130:(* Wait for Finishing movement *)
		IF 	(MoveWorkStored AND WorkPosition) OR
			(MoveInitStored AND InitPosition)	THEN
			WorkingStep:=140;
		END_IF
140:(* Reset Coils if necessary *)
		IF  sInit.KindOfValve='B' AND
			(	( NoOfWorkSensors>0 AND MoveWorkStored) OR
				( NoOfInitSensors>0 AND MoveInitStored) ) THEN
			CoilA:=FALSE;
			CoilB:=FALSE;
			WorkingStep:=1000;
		ELSE
			WorkingStep:=1000;
		END_IF
999: (* State Error *)
		State:=STATE_ERROR;
1000: (* State OK *)
		State:=STATE_OK;
		TimerTimeOut.Start:=FALSE;
		IF 	NOT MoveWork AND	NOT MoveInit OR
			MoveInit AND MoveWorkStored OR
			MoveWork AND MoveInitStored THEN
			WorkingStep:=0;
		END_IF
	END_CASE
	(*--------------------------------------------------------------------
		Handle Timeout
  --------------------------------------------------------------------*)
	IF TimerTimeOut.Timeout THEN
		State:=STATE_TIMEOUT;
		FB_ReadXmlLineMsg.ID:='timeout';
		Error.No:=1;
		Error.Text:=sInit.InstName;
		Error.Text:=CONCAT(Error.Text,': ');
		Error.Text:=CONCAT(Error.Text,sInit.Description);
		Error.Text:=CONCAT(Error.Text,' - ');
		Error.Text:=CONCAT(Error.Text,FB_ReadXmlLineMsg.Text);

		(* Set Flags to Raise Error in ValveSensor Object *)
		IF 	NoOfInitSensors>0 THEN
			FOR IdxInit:=1 TO NoOfInitSensors DO
				ValveInitOut[IdxInit].SignalHiExpected:=MoveInitStored;
				ValveInitOut[IdxInit].SignalLoExpected:=MoveWorkStored;
			END_FOR
		END_IF
		IF 	NoOfWorkSensors>0 THEN
			FOR IdxWork:=1 TO NoOfWorkSensors DO
				ValveWorkOut[IdxWork].SignalHiExpected:=MoveWorkStored;
				ValveWorkOut[IdxWork].SignalLoExpected:=MoveInitStored;
			END_FOR
		END_IF
	ELSE
		(* Reseet Flags to Raise Error in ValveSensor Object *)
		IF 	NoOfInitSensors>0 THEN
			FOR IdxInit:=1 TO NoOfInitSensors DO
				ValveInitOut[IdxInit].SignalHiExpected:=FALSE;
				ValveInitOut[IdxInit].SignalLoExpected:=FALSE;
			END_FOR
		END_IF
		IF 	NoOfWorkSensors>0 THEN
			FOR IdxWork:=1 TO NoOfWorkSensors DO
				ValveWorkOut[IdxWork].SignalHiExpected:=FALSE;
				ValveWorkOut[IdxWork].SignalLoExpected:=FALSE;
			END_FOR
		END_IF
	END_IF
	(*--------------------------------------------------------------------
		Handle unallowed Signalchange without Movecommand
  --------------------------------------------------------------------*)
	IF 	State=State_Wait AND
		NOT sInit.DisableSignalMonitoring THEN
		(* Set Flags to Raise Error in ValveSensor Object *)
		IF  	(MoveInitStored AND NOT InitPosition) OR
			(MoveWorkStored AND NOT WorkPosition)	THEN
			State:=STATE_ERROR;
			FB_ReadXmlLineMsg.ID:='SensorFault';
			Error.No:=1;
			Error.Text:=sInit.InstName;
			Error.Text:=CONCAT(Error.Text,': ');
			Error.Text:=CONCAT(Error.Text,sInit.Description);
			Error.Text:=CONCAT(Error.Text,' - ');
			Error.Text:=CONCAT(Error.Text, FB_ReadXmlLineMsg.Text);

			IF 	NoOfInitSensors>0 THEN
				FOR IdxInit:=1 TO NoOfInitSensors DO
					ValveInitOut[IdxInit].SignalHiExpected:=MoveInitStored;
					ValveInitOut[IdxInit].SignalLoExpected:=MoveWorkStored;
				END_FOR
			END_IF
			IF 	NoOfWorkSensors>0 THEN
				FOR IdxWork:=1 TO NoOfWorkSensors DO
					ValveWorkOut[IdxWork].SignalHiExpected:=MoveWorkStored;
					ValveWorkOut[IdxWork].SignalLoExpected:=MoveInitStored;
				END_FOR
			END_IF
		END_IF

	END_IF
	(*--------------------------------------------------------------------
		Call Timers
  --------------------------------------------------------------------*)
	TimerTimeOut(MTime:=sInit.MaxTime);
	DampBothTimer(PT:=DINT_TO_TIME(sInit.DampBothTime));
	(*--------------------------------------------------------------------
		Updating processtime (if State_RUN, STATE_TIMEOUT, STATE_RESETS, or STATE_STOPPED)
  --------------------------------------------------------------------*)
	IF	(State=State_RUN OR
		State=STATE_TIMEOUT OR
		State=STATE_RESETS OR
		State=STATE_STOPPED) AND
		sInit.MaxTime<>0 AND
		 ( NoOfInitSensors<>0 OR NoOfWorkSensors<>0)	THEN
		ProcessTime:=TimerTimeOut.PTime;
	END_IF
(*--------------------------------------------------------------------
	HomePosition
  --------------------------------------------------------------------*)

IF	sVisu.Description <> '' THEN
	CASE	sInit.HomePosDefine OF

	HOME_INIT:
		HomePosition:=InitPosition AND NOT WorkPosition AND (sInit.KindOfValve<>'2G' OR CoilBState);
	HOME_WORK:
		HomePosition:=WorkPosition AND NOT InitPosition AND (sInit.KindOfValve<>'2G' OR CoilAState);
	HOME_BOTH:
		HomePosition:=WorkPosition OR InitPosition;
	HOME_ALWAYS:
		HomePosition:=TRUE;
	ELSE
		HomePosition:=FALSE;
	END_CASE


(* Generating home position*)
	IF 	NOT HomePosition THEN
		ListHomeNOK(InstName:=sInit.InstName,Description:=FB_ReadXmlLineConf.Text);
	END_IF

	(* Object-homeposition concat with mainhomeposition *)
	gHomeOk:=gHomeOk AND HomePosition;
END_IF
(*------------------------------------------------------------------
	Update Visu
  ------------------------------------------------------------------*)
	sVisu.InstName:=sInit.InstName;

	sVisu.ProcessTime:=ProcessTime;
	sVisu.HomePosition:=HomePosition;
	sVisu.CoilA:=CoilA;
	sVisu.CoilB:=CoilB;
	sVisu.NoOfInitSensors:=NoOfInitSensors;
	sVisu.NoOfWorkSensors:=NoOfWorkSensors;
	sVisu.NoOfValveCoils:=NoOfValveCoils;

	sVisu.SAInitPosName:=SensorInitIn[1].SensorName;
	sVisu.SBInitPosName:=SensorInitIn[2].SensorName;
	sVisu.SCInitPosName:=SensorInitIn[3].SensorName;
	sVisu.SDInitPosName:=SensorInitIn[4].SensorName;
	sVisu.SEInitPosName:=SensorInitIn[5].SensorName;
	sVisu.SAWorkPosName:=SensorWorkIn[1].SensorName;
	sVisu.SBWorkPosName:=SensorWorkIn[2].SensorName;
	sVisu.SCWorkPosName:=SensorWorkIn[3].SensorName;
	sVisu.SDWorkPosName:=SensorWorkIn[4].SensorName;
	sVisu.SEWorkPosName:=SensorWorkIn[5].SensorName;

	sVisu.AInitPosition:=SensorInitIn[1].SensorSignal;
	sVisu.BInitPosition:=SensorInitIn[2].SensorSignal;
	sVisu.CInitPosition:=SensorInitIn[3].SensorSignal;
	sVisu.DInitPosition:=SensorInitIn[4].SensorSignal;
	sVisu.EInitPosition:=SensorInitIn[5].SensorSignal;
	sVisu.AWorkPosition:=SensorWorkIn[1].SensorSignal;
	sVisu.BWorkPosition:=SensorWorkIn[2].SensorSignal;
	sVisu.CWorkPosition:=SensorWorkIn[3].SensorSignal;
	sVisu.DWorkPosition:=SensorWorkIn[4].SensorSignal;
	sVisu.EWorkPosition:=SensorWorkIn[5].SensorSignal;

(*------------------------------------------------------------------
	Reset-Handling
  ------------------------------------------------------------------*)
IF 	Reset THEN
	State:=STATE_RESETS;
	WorkingStep:=0;
	ProcessTime:=0;
	TimerTimeOut.Start:=FALSE;
	DampBothTimer.IN:=FALSE;
	CoilA:=FALSE;
	CoilB:=FALSE;
	MoveWorkStored:=FALSE;
	MoveInitStored:=FALSE;
END_IF

(*------------------------------------------------------------------
	Error-Handling
  ------------------------------------------------------------------*)
ErrorElapsed(CLK:= Error.Text<>'');
IF ErrorElapsed.Q THEN
	Error.DateTime:=gVarDTSystemtime;
END_IF

IF Error.Text<>''	AND ST_Lng.b_EndChangeLng THEN
	Error.Typ:=0;
	(*Error.DateTime:=;*)
	ErrorHandler.AddError(
			ErrorToAdd:=Error,
			sVisu:=Visu.ErrorHandler);
END_IF

IF 	NOT Enable AND ModeSelect.Mode=MODE_MANUAL AND
	Error.Text='' AND strAnlayse<>''THEN

	strAnlayse:=CONCAT(' +++ gesperrt durch : ',strAnlayse);

	LaufschriftAnalyse(
	N:= 40,
	StepWidth:=1,
	PT:= t#100ms ,
	Text:= strAnlayse,
	Display=>sVisu.ErrorString );

	strAnlayse:='';
ELSE
	IF Error.Text<>'' THEN
		TempString:=CONCAT(' --- ',Error.Text);
		LaufschriftObj(
		N:= 40,
		StepWidth:=1,
		PT:= t#100ms ,
		Text:= TempString,
		Display=>sVisu.ErrorString );
	ELSE
		sVisu.ErrorString:='';
	END_IF
END_IF

(*------------------------------------------------------------------
	Reset Inputs
  ------------------------------------------------------------------*)
MoveWork		:=FALSE; 				(* Move to Workposition *)
MoveInit		:=FALSE;				(* Move to Initposition *)
Enable			:=FALSE; 				(* Enables the operations on the valve *)
Reset			:=FALSE; 				(* switch for resetting the object *)

sVisu.InstName:=sInit.InstName;
sVisu.BitName:=sInit.BitName;
sVisu.BtnMoveWork.Text:=sInit.WorkDescription;
sVisu.BtnMoveInit.Text:=sInit.InitDescription;
sVisu.ErrorPresent:=Error.Text<>'';

FB_ReadXmlLineConf(
	Prefix:= 'CONFIG',
	ID:= sInit.InstName,
	File:= 'CONFIG.xml',
	Text=> sVisu.Description );

FB_ReadXmlLineMsg(
	Prefix:= 'MSG',
	ID:= ,
	File:= 'MSG.xml',
	Text=>);


IF 	State = STATE_ERROR THEN
	Error.Text:=sInit.InstName;
	Error.Text:=CONCAT(Error.Text,': ');
	Error.Text:=CONCAT(Error.Text,sInit.Description);
	Error.Text:=CONCAT(Error.Text,' - ');
	Error.Text:=CONCAT(Error.Text,FB_ReadXmlLineMsg.Text);
END_IF
END_FUNCTION_BLOCK
ACTION AddInitSensor:
NoOfInitSensors:=NoOfInitSensors+1;
END_ACTION
ACTION AddWorkSensor:
NoOfWorkSensors:=NoOfWorkSensors+1;
END_ACTION

(* POU System/HelpFunctions/CheckProcTime, ST *)
FUNCTION_BLOCK CheckProcTime
VAR_OUTPUT
	PTime		: DINT;	(* Time since start of the timer *)
	Timeout		: BOOL; (* Flag if Timeout occured *)
END_VAR
VAR_INPUT
	MTime		: DINT;	(* Time to timeout *)
	Start		: BOOL;	(* True starts the Timer, False resets *)
END_VAR
VAR
	TONT		: TON;	(* Timer counting Timer *)
END_VAR
(* Start Timer if Start is True.
Stop Timer ,if Start is false.
Timer maximal counting to two hours. *)
TONT(IN:=Start,PT:=T#2h);

(* Updating the Processtime PTime. You get it if you change the output ET of TONT to DWORD.. *)
PTime:=TIME_TO_DWORD(TONT.ET);

(* Setting output Timeout
No Timeout IF Timer stopped OR mtime > ptime*)
IF 	MTime > PTime OR NOT Start THEN
	Timeout:=FALSE;
ELSE
	Timeout:=TRUE;
END_IF
END_FUNCTION_BLOCK

(* POU zLibrary/_HelpFunctions/FB_Laufschrift, ST *)
FUNCTION_BLOCK FB_Laufschrift
VAR_INPUT
	N 						:INT; (* Max output Stringlength *)
	StepWidth				:INT:=1;
	PT 						:TIME;
	Text 					:STRING; (* Original String *)
END_VAR
VAR_OUTPUT
	Display 					:STRING(255); (* Output String *)
END_VAR
VAR
	delay 					:TP;
	TempOutputString		:STRING(255);
	TempInputText			:STRING(255);
	step 					:INT;
END_VAR
(* generate next ticker when delay is low *)
IF 	N < LEN(text) THEN
	IF 	NOT delay.Q THEN
		(* increase step for next tick *)
		TempInputText:=text;
		step := step + StepWidth;

		IF step > LEN(TempInputText) THEN
			step := 1;
		END_IF

		(* extract dispay from text *)
		TempOutputString := MID(TempInputText, N, step);

		IF 	LEN(TempOutputString)<N THEN
			TempOutputString:=CONCAT(TempOutputString,TempInputText);
			TempOutputString:=LEFT(TempOutputString,N);
			Display:=TempOutputString;
		ELSE
			Display:=TempOutputString;
		END_IF
		(* set delay timer for next tick *)
		delay(IN := TRUE, PT := PT);
	ELSE
		(* execute delay timer *)
		delay(in := FALSE);
	END_IF
ELSE
	display := text;
END_IF
END_FUNCTION_BLOCK

(* POU zLibrary/Valve/FB_ValveSensor, ST *)
FUNCTION_BLOCK FB_ValveSensor
VAR_INPUT
	ValveObject					: POINTER TO FB_Valve;		(* Pointer to declared Valve Instance *)
	sInit							: sValveSensorInit; 				(* Intialisation Informations e.g. Object Name *)
END_VAR
VAR_IN_OUT

END_VAR
VAR_OUTPUT
END_VAR
VAR
	ValveSensor	 			AT %I* :	BOOL; 					(* Sensor A InitPosition *)

	(* Sensor Handling *)
	ValveOut					: sValveSensor_ValveOut; 		(* Signals from Valve Object *)
	SensorOut					: sValveSensor_SensorOut;		(* Signals to Valve Object *)

	ValveSensorNo				: DINT; 							(* Number of Sensor given from ValveObject *)

	sVisuValveDummy			: sValveVisu; 					(* Dummy struct for Calling Action from Valve Object  *)

(* Init Handling *)
	InitState						: BOOL :=	FALSE;				(* Internal State for initialising *)
	InitStep						: INT;							(* Init Step StateMachine *)

(*  Error Handling *)
	Error						: ErrorStruct;						(* Local Error Struct *)
	ErrorElapsed				: R_TRIG;						(* Flag to Store Systemtime in Errorstruct when the error raising *)

	FB_ReadXmlLineConf		: FB_ReadXmlLine;
	FB_ReadXmlLineMsg		: FB_ReadXmlLine;
END_VAR
IF 	NOT InitState THEN
	CASE InitStep OF
	0: (* Init Instance *)
			InitStep:=100;

	100: (* Init Done *)

		IF	ValveSensorNo=0 THEN
			IF sInit.SensorType=sValveSensorType_INIT	THEN
		   		ValveObject^.AddInitSensor(sVisu:=sVisuValveDummy);
				ValveSensorNo:=ValveObject^.NoOfInitSensors;
			ELSE
		   		ValveObject^.AddWorkSensor(sVisu:=sVisuValveDummy);
				ValveSensorNo:=ValveObject^.NoOfWorkSensors;
			END_IF

			SensorOut.SensorName:=sInit.BitName;
			SensorOut.SensorType:=sInit.SensorType;

		END_IF

		InitState:=TRUE;
	END_CASE


ELSE
	(* Init State OK *)
	Error.No:=0;
	Error.Text:='';

	IF 	sInit.SensorType=sValveSensorType_INIT	THEN
		ValveOut:=ValveObject^.ValveInitOut[ValveSensorNo];
	ELSE
		ValveOut:=ValveObject^.ValveWorkOut[ValveSensorNo];
	END_IF

	(* Generate Errors  *)

	(* Check Signal Hi *)
	IF 	ValveOut.SignalHiExpected AND
		NOT ValveSensor	THEN
	  	Error.No:=1;
(*		Error.Text:=CONCAT(ValveObject^.sInit.InstName,' - ');*)
		FB_ReadXmlLineMsg.ID:='SensorFaultNotHigh';
		Error.Text:=CONCAT(Error.Text,sInit.InstName);
		Error.Text:=CONCAT(Error.Text,' :');
		Error.Text:=CONCAT(Error.Text,FB_ReadXmlLineConf.Text);
		Error.Text:=CONCAT(Error.Text,' - ');
		Error.Text:=CONCAT(Error.Text,FB_ReadXmlLineMsg.Text);

	END_IF


	(* Check Signal Low *)
	IF 	ValveOut.SignalLoExpected AND
		ValveSensor THEN
	  	Error.No:=1;
(*		Error.Text:=CONCAT(ValveObject^.sInit.InstName,' - ');*)
		FB_ReadXmlLineMsg.ID:='SensorFaultNotLow';
		Error.Text:=CONCAT(Error.Text,sInit.InstName);
		Error.Text:=CONCAT(Error.Text,' :');
		Error.Text:=CONCAT(Error.Text,FB_ReadXmlLineConf.Text);
		Error.Text:=CONCAT(Error.Text,' - ');
		Error.Text:=CONCAT(Error.Text,FB_ReadXmlLineMsg.Text);
	END_IF

	(* Write Sensor stete in local out Structure *)
	SensorOut.SensorSignal:=ValveSensor;

	(* Give local "out structure" to Valve object *)
	IF 	sInit.SensorType=sValveSensorType_INIT THEN
		ValveObject^.SensorInitIn[ValveSensorNo]:=SensorOut;
	ELSE
		ValveObject^.SensorWorkIn[ValveSensorNo]:=SensorOut;
	END_IF

END_IF

(*------------------------------------------------------------------
	Error-Handling
  ------------------------------------------------------------------*)

ErrorElapsed(CLK:= Error.Text<>'');
IF 	ErrorElapsed.Q THEN
	Error.DateTime:=gVarDTSystemtime;
END_IF

IF Error.Text<>''	AND ST_Lng.b_EndChangeLng THEN
	Error.Typ:=0;
	ErrorHandler.AddError(
				ErrorToAdd:=Error,
				sVisu:=Visu.ErrorHandler);
END_IF

(*------------------------------------------------------------------
	Language-Handling
  ------------------------------------------------------------------*)

FB_ReadXmlLineConf(
	Prefix:= 'CONFIG',
	ID:= sInit.InstName,
	File:= 'CONFIG.xml',
	Text=> );


FB_ReadXmlLineMsg(
	Prefix:= 'MSG',
	ID:= ,
	File:= 'MSG.xml',
	Text=>);

IF 	Error.Text<>'' THEN
	Error.Text:=CONCAT(Error.Text,sInit.InstName);
	Error.Text:=CONCAT(Error.Text,' :');
	Error.Text:=CONCAT(Error.Text,FB_ReadXmlLineConf.Text);
	Error.Text:=CONCAT(Error.Text,' - ');
	Error.Text:=CONCAT(Error.Text,FB_ReadXmlLineMsg.Text);
END_IF
END_FUNCTION_BLOCK

(* POU zLibrary/AnaIn/FB_AnaInDint, ST *)
FUNCTION_BLOCK FB_AnaInDint
VAR_INPUT
	sInit					:sAnaInInit;	(* Initializingvalues to the Instance *)
END_VAR
VAR_OUTPUT
	State					:StateObject;	(* State of the object *)
	HomePosition			:BOOL;			(* object in home-position*)
	Value					:REAL;
END_VAR
VAR_IN_OUT
	sVisu					:sAnaInVisu;
END_VAR
VAR
	AnaInValue		AT %I* 	:DINT;			(* Ana in value *)

	Error					:ErrorStruct;
	TempErrorText			:STRING(255);
	InitState				:BOOL:=FALSE;	(* Internal State for initialising *)

	diffSource				:REAL;
	diffTarget				:REAL;

	FB_ReadXmlLineConf		:FB_ReadXmlLine;
	FB_ReadXmlLineMsg		:FB_ReadXmlLine;
END_VAR
Error.No:=0;
Error.Text:='';

(*------------------------------------------------------------------
	Initialization
  ------------------------------------------------------------------*)
IF  NOT InitState THEN
	InitState:=TRUE;

	(* Check instance name *)
	IF sInit.InstName=''THEN
		InitState:=FALSE;
		State:=STATE_ERROR;
		FB_ReadXmlLineMsg.ID:='InstNameNotDefined';

		TempErrorText:=sInit.BitInName;
		TempErrorText:=CONCAT(TempErrorText,' :');
		TempErrorText:=CONCAT(TempErrorText,sVisu.Description);
  		TempErrorText:=CONCAT(TempErrorText,' -> ');
		TempErrorText:=CONCAT(TempErrorText,FB_ReadXmlLineMsg.Text);
		Error.No:=4;
		(*Error.Text:='InstName not defined';*)
	(*CheckDescription*)
	ELSIF
		sInit.Description=''THEN
		InitState:=FALSE;
		State:=STATE_ERROR;
		FB_ReadXmlLineMsg.ID:='DescriptionNotDefined';

		TempErrorText:=sInit.BitInName;
		TempErrorText:=CONCAT(TempErrorText,' :');
		TempErrorText:=CONCAT(TempErrorText,sVisu.Description);
  		TempErrorText:=CONCAT(TempErrorText,' -> ');
		TempErrorText:=CONCAT(TempErrorText,FB_ReadXmlLineMsg.Text);
		Error.No:=4;
		(*Error.Text:='Description not defined';*)
	END_IF

	sVisu.InstName		:= sInit.InstName;
	sVisu.Description	:= sInit.Description;
	sVisu.ErrorString	:= Error.Text;
END_IF

(* Add InitState to Global-Init-State to collect all Objects *)
gInitCollect:=gInitCollect AND InitState;

IF 	InitState THEN
	diffSource := sinit.ScalingSensorValueMax - sinit.ScalingSensorValueMin;
  	diffTarget := sinit.ScalingOutputValueMax - sinit.ScalingOutputValueMin;
 	(*Value := (((AnaInValue-sinit.ScalingOutputValueMin)/diffSource)*diffTarget)+sinit.ScalingOutputValueMin;*)
 	Value :=  (AnaInValue- sinit.ScalingSensorValueMin) / (diffSource  / diffTarget) ;

	sVisu.AnaInValue:=Value;

END_IF
(* ------------------------------------------------------------------------------------------ *)
(* ---------------- LANGUAGE auslesen aus der XML Datei-------- *)
(* ------------------------------------------------------------------------------------------ *)
sVisu.BitInName:=sInit.BitInName;
sVisu.InstName:=sInit.InstName;
sVisu.ErrorPresent:=Error.Text<>'';

FB_ReadXmlLineConf(
	Prefix:= 'CONFIG',
	ID:= sInit.InstName,
	File:= 'CONFIG.xml',
	Text=> sVisu.Description  );


FB_ReadXmlLineMsg(
	Prefix:= 'MSG',
	ID:= ,
	File:= 'MSG.xml',
	Text=>);

IF 	State = STATE_ERROR THEN
	TempErrorText:=sInit.BitInName;
	TempErrorText:=CONCAT(TempErrorText,' :');
	TempErrorText:=CONCAT(TempErrorText,sVisu.Description);
	TempErrorText:=CONCAT(TempErrorText,' -> ');
	TempErrorText:=CONCAT(TempErrorText,FB_ReadXmlLineMsg.Text);
END_IF
END_FUNCTION_BLOCK

(* POU zLibrary/AnaIn/FB_Encoder, ST *)
FUNCTION_BLOCK FB_Encoder
VAR_INPUT
	sInit					:sEncoderInit;	(* Initializingvalues to the Instance *)
	Reset					:BOOL;
END_VAR
VAR_OUTPUT
	State					:StateObject;	(* State of the object *)
	rpmValue			: LREAL;		(* rpm *)
	posValue			: LREAL;		(* mm *)
	Drehrichtung		: enum_Drehrichtung;
END_VAR
VAR_IN_OUT
	sVisu				:sEncoderVisu;
END_VAR
VAR

	Error					:ErrorStruct;
	TempErrorText			:STRING(255);
	ErrorElapsed			:BOOL;
	LaufschriftErrh			:FB_Laufschrift;
	LaufschriftObj			:FB_Laufschrift_STR255;
	InitState				:BOOL:=FALSE;	(* Internal State for initialising *)



	FB_ReadXmlLineConf		:FB_ReadXmlLine;
	FB_ReadXmlLineMsg		:FB_ReadXmlLine;
END_VAR


(*==================================================================*)
VAR_OUTPUT

END_VAR

VAR
	fb_ton_Reset		: TON;
	fb_ton_steht		: TON;
	fb_ton_dreht		: TON;

	fb_rTrigReset		: R_TRIG;
	fb_rTrigUnderflow		: R_TRIG;
	fb_rTrigOverflow		: R_TRIG;

	i_count_ueberlauf		: DINT;		(* +- 64bit *)
	lr_xBit		: LREAL;
	lr_rpmHelp	: LREAL;	(*°*)

	
	e_Value					AT %I* : UINT;		(* 65535 *)
	e_CountUnderflow		AT %I* : BOOL;
	e_CountOverflow			AT %I* : BOOL;
	a_CountReset			AT %Q* : BOOL;

END_VAR
VAR CONSTANT



END_VAR
Error.No:=0;
Error.Text:='';

(*------------------------------------------------------------------
	Initialization
  ------------------------------------------------------------------*)
IF  NOT InitState THEN
	InitState:=TRUE;
	State:=STATE_OK;
	(* Check instance name *)
	IF 	sInit.InstName=''THEN
		InitState:=FALSE;
		State:=STATE_ERROR;
		FB_ReadXmlLineMsg.ID:='InstNameNotDefined';

		TempErrorText:=sInit.BitInName;
		TempErrorText:=CONCAT(TempErrorText,' :');
		TempErrorText:=CONCAT(TempErrorText,sVisu.Description);
  		TempErrorText:=CONCAT(TempErrorText,' -> ');
		TempErrorText:=CONCAT(TempErrorText,FB_ReadXmlLineMsg.Text);
		Error.No:=4;
	(*CheckDescription*)
	ELSIF
		sInit.Description=''THEN
		InitState:=FALSE;
		State:=STATE_ERROR;
		FB_ReadXmlLineMsg.ID:='DescriptionNotDefined';

		TempErrorText:=sInit.BitInName;
		TempErrorText:=CONCAT(TempErrorText,' :');
		TempErrorText:=CONCAT(TempErrorText,sVisu.Description);
  		TempErrorText:=CONCAT(TempErrorText,' -> ');
		TempErrorText:=CONCAT(TempErrorText,FB_ReadXmlLineMsg.Text);
		Error.No:=4;
	ELSIF
		sInit.i_InkProRpm=0THEN
		InitState:=FALSE;
		State:=STATE_ERROR;
		FB_ReadXmlLineMsg.ID:='InkProRpmNotDefined';

		TempErrorText:=sInit.BitInName;
		TempErrorText:=CONCAT(TempErrorText,' :');
		TempErrorText:=CONCAT(TempErrorText,sVisu.Description);
  		TempErrorText:=CONCAT(TempErrorText,' -> ');
		TempErrorText:=CONCAT(TempErrorText,FB_ReadXmlLineMsg.Text);
		Error.No:=4;
	END_IF

END_IF

(* Add InitState to Global-Init-State to collect all Objects *)
gInitCollect:=gInitCollect AND InitState;

(*==================================================================*)
IF  InitState THEN
	(* Drehrichtung ermitteln *)
	fb_ton_steht(PT:=T#50MS);
	IF	lr_rpmHelp > rpmValue - 0.0001 AND
		lr_rpmHelp < rpmValue + 0.0001 THEN
		fb_ton_steht.IN:=TRUE;
		IF	fb_ton_steht.Q THEN
			Drehrichtung:= STEHT;
		END_IF
	ELSIF
		lr_rpmHelp < rpmValue THEN
		fb_ton_steht.IN:=FALSE;
		Drehrichtung:= VORWAERTS;
	ELSIF
		lr_rpmHelp > rpmValue THEN
		fb_ton_steht.IN:=FALSE;
		Drehrichtung:= RUECKWAERTS;
	END_IF
	lr_rpmHelp:=rpmValue;
	
	(* Encoderüberlauf*)
	fb_rTrigUnderflow(CLK:= e_CountUnderflow);
	fb_rTrigOverflow(CLK:= e_CountOverflow);
	IF 	fb_rTrigUnderflow.Q THEN
		i_count_ueberlauf:=i_count_ueberlauf - 1;
	ELSIF
		fb_rTrigOverflow.Q THEN
		i_count_ueberlauf:=i_count_ueberlauf + 1;
	END_IF

	(* bei Reset Nullen *)
	fb_ton_Reset(IN:=Reset , PT:= T#300MS , Q=> , ET=> );
	a_CountReset:=Reset OR sVisu.Reset;
	fb_rTrigReset(CLK:=fb_ton_Reset.Q, );
	IF	fb_rTrigReset.Q THEN
		Reset:=FALSE;
	END_IF

	(* aktuelle Position *)
	IF	e_Value <> 0 THEN
		lr_xBit:=EXPT(2,16);												(* 16 bit=65535  Inkremente Encoder*)
		rpmValue:= e_Value + (lr_xBit * DINT_TO_LREAL(i_count_ueberlauf));	(* Inkremente*)
		rpmValue:= rpmValue / sInit.i_InkProRpm;							(* Umdrehungen in Grad*)
	ELSE
		rpmValue:= 0;
		i_count_ueberlauf:=0;
	END_IF
	IF	sInit.lr_LaengeProRpm > 0 THEN
		posValue:= rpmValue * sInit.lr_LaengeProRpm;					(* Strecke in mm*)
	ELSE
		posValue:= 0;													(* Strecke in mm*)
	END_IF

	sVisu.posValue:=posValue;
	sVisu.rpmValue:=rpmValue;
	sVisu.Drehrichtung:=Drehrichtung;
END_IF
(* ------------------------------------------------------------------------------------------ *)
(* ---------------- LANGUAGE auslesen aus der XML Datei-------- *)
(* ------------------------------------------------------------------------------------------ *)
sVisu.BitInName:=sInit.BitInName;
sVisu.InstName:=sInit.InstName;
sVisu.ErrorPresent:=Error.Text<>'';

(*  *)
IF 	State=STATE_ERROR AND
	NOT ErrorElapsed THEN
	ErrorElapsed:=TRUE;
	Error.DateTime:=gVarDTSystemtime;
ELSIF
	State<>STATE_ERROR THEN
	ErrorElapsed:=FALSE;
	TempErrorText:='';
END_IF;

IF 	Error.Text<>'' AND
	ST_Lng.b_EndChangeLng THEN
	(*Error.DateTime:=;*)
	Error.Typ:=0;
	ErrorHandler.AddError(ErrorToAdd:=Error,
	sVisu:=Visu.ErrorHandler);
END_IF


FB_ReadXmlLineConf(
	Prefix:= 'CONFIG',
	ID:= sInit.InstName,
	File:= 'CONFIG.xml',
	Text=> sVisu.Description  );

FB_ReadXmlLineMsg(
	Prefix:= 'MSG',
	ID:= ,
	File:= 'MSG.xml',
	Text=>);

IF 	State = STATE_ERROR THEN
	TempErrorText:=sInit.BitInName;
	TempErrorText:=CONCAT(TempErrorText,' :');
	TempErrorText:=CONCAT(TempErrorText,sVisu.Description);
	TempErrorText:=CONCAT(TempErrorText,' -> ');
	TempErrorText:=CONCAT(TempErrorText,FB_ReadXmlLineMsg.Text);
END_IF


LaufschriftErrh(
N:= 160,
StepWidth:=1,
PT:= t#100ms ,
Text:= TempErrorText,
Display=>Error.Text );

LaufschriftObj(
N:= 40,
StepWidth:=1,
PT:= t#100ms ,
Text:= TempErrorText,
Display=>sVisu.ErrorString );
END_FUNCTION_BLOCK

(* POU zLibrary/DigIn/FB_DigIn, ST *)
FUNCTION_BLOCK FB_DigIn

VAR_OUTPUT
	State						: StateObject;	(* State of the object *)
	HomePosition				: BOOL;			(* object in home-position*)
	SignalIn						: BOOL;			(* Static signal of digital input *)
	SignalInDelayed				: BOOL;			(* Static signal of digital input but with on and of delay times *)
END_VAR
VAR_INPUT
	CheckSignalHigh			: BOOL;		 	(* Signal check  HIGH *)
	CheckSignalLow			: BOOL;		 	(* Signal check  LOW  *)

	Reset						: BOOL;			(* switch for resetting the control *)

	SFCCurrentStep				: STRING(40);	(* aktually step in the order of events *)
	SFCCurrentPOU				: STRING(40);	(* Name of the order of events*)

	sInit						: sDigInInit;		(* Initializingvalues to the Instance *)
END_VAR
VAR_IN_OUT
	sVisu						: sDigInVisu;
END_VAR
VAR
	BitInToCheck				AT %I* :BOOL;		(* Bit input signal to check *)

	ProcessTime					: DINT;					(* Counts the time in steps of 100ms since starting operation *)

	TimerTimeOut				: CheckProcTime;		(* Timer generates timeout signal *)
	Error						: ErrorStruct;
	ErrorElapsed				: BOOL;
	TempErrorText				: STRING(255);
	HomePositionInfo			: DINT;							(* missing to home posistion *)
	ResetIntern					: BOOL;							(* Internal reset signal *)


	BtnReset					: VisuButton;			(* Manage button *)

	StateOK_CycleFlag			: BOOL;

	FirstCheckCycle				:  R_TRIG;

	IputOnDelayTime				: TON;
	IputOffDelayTime			: TOF;

	(* --------------------------------------------------------------------------------- *)
	(*         Internal Variables	Visu				                                           *)
	(* --------------------------------------------------------------------------------- *)
	LaufschriftErrh				:FB_Laufschrift;
	LaufschriftObj				:FB_Laufschrift;

	FB_ReadXmlLineConf		:FB_ReadXmlLine;
	FB_ReadXmlLineMsg		:FB_ReadXmlLine;

END_VAR
Error.No:=0;
Error.Text:='';
TempErrorText:='';

(*------------------------------------------------------------------
	Initialization
  ------------------------------------------------------------------*)


(* Add InitState to Global-Init-State to collect all Objects *)
gInitCollect:=gInitCollect ;

IF gInitOk THEN

StateOK_CycleFlag := State=State_ok;


(*------------------------------------------------------------------
	Show and Read Buttons
  ------------------------------------------------------------------*)

BtnReset(	Button:=sVisu.BtnReset,
					Enable:=TRUE ,
					Visible:=ModeSelect.Mode=MODE_MANUAL,
					TextOn:='Reset',
					TextOff:='Reset',
					PressedExt:=FALSE ,
					StateOn:= FALSE ,
					);

	(*------------------------------------------------------------------
	Manual-Mode
  ------------------------------------------------------------------*)
	IF  ModeSelect.Mode=MODE_MANUAL THEN

		SFCCurrentStep:=sInit.InstName;
		SFCCurrentPOU:='MODE_MANUAL';
	END_IF (*ModeSelect.Mode=MODE_MANUAL*)


	(*reset timer in first cycle of checking*)
	FirstCheckCycle(CLK := CheckSignalHigh OR CheckSignalLow );

	IF 	FirstCheckCycle.Q THEN
		ProcessTime:=TimerTimeOut.PTime;
	END_IF

	(*------------------------------------------------------------------
	Mode higher manual mode (auto, tip or homeposrun)
  ------------------------------------------------------------------*)
	 	IF	( ModeSelect.Mode>MODE_MANUAL OR sInit.EnableInEveryMode) AND
			( CheckSignalHigh OR CheckSignalLow )	THEN

		(* Check input signal                                      *)
		(*=========================================================*)

		(* Check signal low and input is low*)
		IF 	NOT BitInToCheck AND
			CheckSignalLow AND
			NOT CheckSignalHigh THEN
			(* Check input low and it is low *)
			TimerTimeOut(Start := FALSE, MTime := (sInit.MaxTime));
			State:=State_OK;

		(* Check input low and input is high*)
		ELSIF
			BitInToCheck AND
			CheckSignalLow AND
			NOT CheckSignalHigh THEN
			TimerTimeOut(Start := TRUE, MTime := (sInit.MaxTime));
			State:=STATE_RUN;
		(* Check input high *)
		ELSIF
			BitInToCheck AND
			NOT CheckSignalLow AND
			CheckSignalHigh THEN
			TimerTimeOut(Start := FALSE, MTime := (sInit.MaxTime));
			State:=State_OK;

		(* Check signal high and input is low*)
		ELSIF
			NOT  BitInToCheck AND
			NOT CheckSignalLow AND
			CheckSignalHigh	THEN
			TimerTimeOut(Start := TRUE, MTime := (sInit.MaxTime));
			State:=STATE_RUN;
		ELSE
			TimerTimeOut(Start := FALSE, MTime := (sInit.MaxTime));

			IF	NOT CheckSignalHigh AND
				NOT CheckSignalLow THEN
				State:=STATE_WAIT;
			END_IF
		END_IF

		(* Timeout check high *)
		IF	TimerTimeOut.Timeout AND
			NOT ResetIntern AND
			State=STATE_RUN AND
			NOT CheckSignalLow AND
			CheckSignalHigh THEN

			State:=STATE_ERROR;
			FB_ReadXmlLineMsg.ID:='SensorFaultNotHigh';

			TempErrorText:=sInit.BitInName;
			TempErrorText:=CONCAT(TempErrorText,' :');
			TempErrorText:=CONCAT(TempErrorText,sVisu.Description);
      			TempErrorText:=CONCAT(TempErrorText,' -> ');
			TempErrorText:=CONCAT(TempErrorText,FB_ReadXmlLineMsg.Text);
			Error.No:=3;
		END_IF
		(* Timeout check low *)
		IF	TimerTimeOut.Timeout AND
			NOT ResetIntern AND
			State=STATE_RUN AND
			CheckSignalLow AND
			NOT CheckSignalHigh THEN
			State:=STATE_ERROR;
			FB_ReadXmlLineMsg.ID:='SensorFaultNotLow';

			TempErrorText:=sInit.BitInName;
			TempErrorText:=CONCAT(TempErrorText,' :');
			TempErrorText:=CONCAT(TempErrorText,sVisu.Description);
      		TempErrorText:=CONCAT(TempErrorText,' -> ');
			TempErrorText:=CONCAT(TempErrorText,FB_ReadXmlLineMsg.Text);
			Error.No:=4;
		END_IF

	ELSE	(* No action *)
		(* Reset ok signal*)
		IF 	State = State_OK AND
			StateOK_CycleFlag THEN
			State:=STATE_WAIT;
		END_IF

	END_IF

END_IF	(* Init ok *)

(*--------------------------------------------------------------------
	Updating processtime (if State_RUN, STATE_ERROR, STATE_RESETS, or STATE_STOPPED)
--------------------------------------------------------------------*)
IF	(State=State_RUN OR
	State=STATE_ERROR OR
	State=STATE_RESETS OR
	State=STATE_STOPPED) AND
	sInit.MaxTime<>0 THEN
	TimerTimeout;
	ProcessTime:=TimerTimeout.PTime;
END_IF

(*------------------------------------------------------------------
	Reset-Handling
  ------------------------------------------------------------------*)
ResetIntern:= 	Reset OR
				BtnReset.Pressed OR
			 	(	State = STATE_ERROR AND
					NOT CheckSignalLow AND
					CheckSignalHigh AND
					BitInToCheck ) OR

			 	(	State = STATE_ERROR AND
					CheckSignalLow AND
					NOT CheckSignalHigh AND
					NOT BitInToCheck) OR

			 	(	State = STATE_ERROR AND
					NOT CheckSignalLow AND
					NOT CheckSignalHigh);

IF 	ResetIntern THEN
	TimerTimeout (Start := FALSE, MTime := (sInit.MaxTime));
	State:= STATE_RESETS;
ELSE
	IF 	State=STATE_RESETS THEN
		State:=STATE_WAIT;
	END_IF
END_IF

(*------------------------------------------------------------------
	Clear all input variables
  ------------------------------------------------------------------*)
Reset:= FALSE;
CheckSignalLow:= FALSE;
CheckSignalHigh:= FALSE;

(*------------------------------------------------------------------
	HomePosition
  ------------------------------------------------------------------*)
HomePositionInfo:=State_OK;

(* Check input signal *)
IF	sInit.HomePosSignal=0 AND
	BitInToCheck THEN
	HomePositionInfo:=11;
END_IF
IF	sInit.HomePosSignal=1 AND
	NOT BitInToCheck THEN
	HomePositionInfo:=10;
END_IF

(* Generating home position*)
(* Zuweisung der Grundstellung*)
IF 	HomePositionInfo=State_OK THEN
	HomePosition:= TRUE;
ELSE
	HomePosition:= FALSE;
	ListHomeNOK(InstName:=sVisu.InstName,Description:=sVisu.Description);
END_IF

(* Objekt-Grundstellung verknüpfen mit GesamtGrundstellung *)
(* object-homeposition concat with mainhomeposition *)
gHomeOk:=gHomeOk AND HomePosition;

(*------------------------------------------------------------------
	Set Visu-Vars
  ------------------------------------------------------------------*)
sVisu.BitInName				:=	sInit.BitInName;
sVisu.BitInToCheck			:=	BitInToCheck;
sVisu.State					:=	State;
sVisu.HomePosition			:=	HomePosition;


(*Copy input-signal to output-var*)
SignalIn:=BitInToCheck;


	(* -------------------------------------------------------------- *)
	(* ------------------ Handle Delay Output --------- *)
	(* -------------------------------------------------------------- *)

	IputOnDelayTime 	(IN := BitInToCheck, PT := DINT_TO_TIME(sInit.IputOnDelayTime));
	IputOffDelayTime 	(IN := BitInToCheck, PT := DINT_TO_TIME(sInit.IputOffDelayTime));

	SignalInDelayed	:=  IputOnDelayTime.Q  OR (IputOffDelayTime.Q AND NOT BitInToCheck);

(*------------------------------------------------------------------
	Error-Handling
  ------------------------------------------------------------------*)
	LaufschriftObj(
	N:= 40,
	StepWidth:=1,
	PT:= t#100ms ,
	Text:= TempErrorText,
	Display=>sVisu.ErrorString );

	LaufschriftErrh(
	N:= 160,
	StepWidth:=1,
	PT:= t#100ms ,
	Text:= TempErrorText,
	Display=>Error.Text );

(*  *)
IF State=STATE_ERROR AND
	NOT ErrorElapsed THEN
	ErrorElapsed:=TRUE;
	Error.DateTime:=gVarDTSystemtime;
END_IF

IF 	State<>STATE_ERROR THEN
	ErrorElapsed:=FALSE;
	TempErrorText:='';
END_IF;

sVisu.ProcessTime:=ProcessTime;

IF 	Error.Text<>''	AND ST_Lng.b_EndChangeLng THEN
	Error.Typ:=0;
	ErrorHandler.AddError(ErrorToAdd:=Error,
	sVisu:=Visu.ErrorHandler);
END_IF

(* ------------------------------------------------------------------------------------------ *)
(* ---------------- LANGUAGE auslesen aus der XML Datei-------- *)
(* ------------------------------------------------------------------------------------------ *)
sVisu.BitInName:=sInit.BitInName;
sVisu.InstName:=sInit.InstName;
sVisu.ErrorPresent:=Error.Text<>'';

FB_ReadXmlLineConf(
	Prefix:= 'CONFIG',
	ID:= sInit.InstName,
	File:= 'CONFIG.xml',
	Text=> sVisu.Description  );


FB_ReadXmlLineMsg(
	Prefix:= 'MSG',
	ID:= ,
	File:= 'MSG.xml',
	Text=>);

IF 	State = STATE_ERROR THEN
	TempErrorText:=sInit.BitInName;
	TempErrorText:=CONCAT(TempErrorText,' :');
	TempErrorText:=CONCAT(TempErrorText,sVisu.Description);
	TempErrorText:=CONCAT(TempErrorText,' -> ');
	TempErrorText:=CONCAT(TempErrorText,FB_ReadXmlLineMsg.Text);
END_IF
END_FUNCTION_BLOCK

(* POU zLibrary/DigOutIn/FB_DigOutIn, ST *)
FUNCTION_BLOCK FB_DigOutIn (*Version 1.2, 20.NOV 2010*)
VAR_OUTPUT
	State					: StateObject;	(* State of the object *)
	HomePosition			: BOOL;					(* object in home-position*)
	SignalOut				: BOOL;							(* Static signal of digital output *)
	SignalIn				: BOOL;							(* Static signal of digital input *)
END_VAR
VAR_INPUT
	SetSignalHigh			: BOOL;		 		 	(* Signal set  HIGH *)
	SetSignalLow			: BOOL;		 			(* Signal set  LOW  *)

	PulseOn					: BOOL;		 			(* Signal pulse On *)
	PulseTime				: DINT; 				(* Length in ms for output impulse *)

	FlashSignal				: BOOL;		 			(* Signal FLASH  *)
	OnTime					: DINT; 				(* In ms for ON time *)
	OffTime					: DINT; 				(* In ms for OFF time *)

	CheckSignalHigh			: BOOL;		 		 	(* Signal check  HIGH *)
	CheckSignalLow			: BOOL;		 			(* Signal check  LOW  *)

	Enable					: BOOL:=TRUE; 	(* Enables the operations on the class *)
	Reset					: BOOL;					(* switch for resetting the control *)

	SFCCurrentStep			: STRING(40);		(* aktually step in the order of events *)
	SFCCurrentPOU			: STRING(40);		(* Name of the order of events*)

	sInit					: sDigOutInInit;		(* Initializingvalues to the Instance *)
	strAnlayse				: STRING(255);  (*String to analyse Lockings*)
END_VAR
VAR_IN_OUT
	sVisu					: sDigOutInVisu;
END_VAR
VAR
	BitOutToSet				AT %Q* :BOOL;		(* Bit output signal to set *)
	BitInToCheck			AT %I* :BOOL;		(* Bit input signal to check *)

	ProcessTime				: DINT;					(* Counts the time in steps of 100ms since starting operation *)

	TimerTimeOut			: CheckProcTime;		(* Timer generates timeout signal *)
	Error					: ErrorStruct;
	ErrorElapsed			: R_TRIG;
	LaufschriftErrh			: FB_Laufschrift;
	LaufschriftObj			: FB_Laufschrift_STR255;
	LaufschriftAnalyse		: FB_Laufschrift_STR255;
	TempString				: STRING(255);

	TempErrorText			: STRING(255);
	OutputAvailable			: BOOL;
	InputAvailable			: BOOL;
	HomePositionInfo		: DINT;							(* missing to home posistion *)
	ResetIntern				: BOOL;							(* Internal reset signal *)
	InitState				: BOOL :=FALSE;		(* Internal State for initialising *)

	BtnOutput				: VisuButton;			(* Manage button *)
	BtnReset				: VisuButton;			(* Manage button *)

	SetOutPulse				: TP;							(* Timer for set output pulse *)
	SetOutPulseActive		: BOOL;
	TimerOn		 			: TON;						(* Timer for output on time *)
	TimerOff		 		: TOF;						(* Timer for output off time *)
  	StateOK_CycleFlag		: BOOL;

	FB_ReadXmlLineConf		: FB_ReadXmlLine;
	FB_ReadXmlLineMsg		: FB_ReadXmlLine;

END_VAR
VAR CONSTANT
	INPUT_CHECKLOW			: DINT:=  21;	(* State input check low *)
	INPUT_CHECKHIGH			: DINT:=  22;	(* State input check  high *)
END_VAR
Error.No:=0;
Error.Text:='';

(*------------------------------------------------------------------
	Initialization
  ------------------------------------------------------------------*)
IF 	NOT InitState THEN
	InitState:=TRUE;

	(* Check instance name *)
	IF 	sInit.InstName='' THEN
		InitState:=FALSE;
		State:=STATE_ERROR;
		Error.No:=4;
		TempErrorText:='InstName not defined';

	(* Check input name *)
	ELSIF
		sInit.BitOutName='' AND  sInit.BitInName='' THEN

		InitState:=FALSE;
		State:=STATE_ERROR;
		Error.No:=4;
		TempErrorText:='No bit out and in name defined';
		sInit.BitOutName:='No output name!';
		sInit.BitInName:='No input name!';
	END_IF

	(* Check output name *)
	IF 	sInit.BitOutName<>'' THEN
		OutputAvailable:=TRUE;
	ELSE
		OutputAvailable:=FALSE;
		sInit.BitOutName:='No output name!';
	END_IF

	(* Check input name *)
	IF 	sInit.BitInName<>'' 	THEN
		InputAvailable:=TRUE;
	ELSE
		InputAvailable:=FALSE;
		sInit.BitInName:='No input name!';
	END_IF

	(* send names to Visu *)
	sVisu.InstName	:= sInit.InstName;
	sVisu.Description	:= sInit.Description;
	sVisu.BitOutName	:= sInit.BitOutName;
	sVisu.InputAvailable	:= InputAvailable;
	sVisu.OutputAvailable	:= OutputAvailable;

END_IF

(* Add InitState to Global-Init-State to collect all Objects *)
gInitCollect:=gInitCollect AND InitState;

IF gInitOk THEN
StateOK_CycleFlag := NOT (State<>State_ok);

(*------------------------------------------------------------------
	Show and Read Buttons
  ------------------------------------------------------------------*)
	BtnOutput(Button:=sVisu.BtnOutput,
						Enable:=(ModeSelect.Mode=MODE_MANUAL OR sInit.EnableVisuInEveryMode ) AND Enable AND OutputAvailable  ,
						Visible:= OutputAvailable,
						TextOn:=sInit.BitOutName,
						TextOff:=sInit.BitOutName,
						PressedExt:=FALSE ,
						StateOn:= FALSE ,
						);

	(*------------------------------------------------------------------
	Manual-Mode
  ------------------------------------------------------------------*)
	IF  	ModeSelect.Mode=MODE_MANUAL OR
		sInit.EnableVisuInEveryMode THEN
		(* Set or reset output manual *)
		IF	BtnOutput.PressedFlag AND
			OutputAvailable AND
			Enable	THEN
			IF 	NOT BitOutToSet THEN
				BitOutToSet:=TRUE;
			ELSE
				BitOutToSet:=FALSE;
			END_IF
		END_IF

		SFCCurrentStep:=sInit.InstName;
		SFCCurrentPOU:='MODE_MANUAL';
	END_IF (*ModeSelect.Mode=MODE_MANUAL*)

	(*------------------------------------------------------------------
	Mode higher manual mode (auto, tip or homeposrun)
  ------------------------------------------------------------------*)
	IF 		(ModeSelect.Mode>MODE_MANUAL OR sInit.EnableInEveryMode OR sInit.EnableVisuInEveryMode) AND
			(	SetSignalHigh OR
				 SetSignalLow OR
				 PulseOn OR
				 SetOutPulseActive OR
				 FlashSignal OR
				 CheckSignalHigh OR
				 CheckSignalLow 	) THEN
	
		(* Set output on off                                       *)
		(*=========================================================*)

		(* Set output signal *)
		IF	SetSignalHigh AND
			NOT SetSignalLow AND
			NOT PulseOn AND
			NOT FlashSignal AND
			OutputAvailable THEN

			BitOutToSet:=TRUE;

			(* If no sensor check then state ok *)
			IF 	NOT InputAvailable	OR
				( NOT CheckSignalHigh AND
				  NOT CheckSignalLow )	THEN

				State:=STATE_OK;
			END_IF
		END_IF
		
		(* Reset output signal *)
		IF	NOT SetSignalHigh AND
			SetSignalLow AND
			NOT PulseOn AND
			NOT FlashSignal AND
			OutputAvailable 	THEN

			BitOutToSet:=FALSE;

			(* If no sensor check then state ok *)
			IF 	NOT InputAvailable OR
				( NOT CheckSignalHigh AND
				  NOT CheckSignalLow )	THEN

				State:=STATE_OK;
			END_IF
		END_IF

		(* Set output with pulse time                              *)
		(*=========================================================*)
		IF	PulseOn OR SetOutPulseActive AND
			OutputAvailable AND
			PulseTime>0 AND
			NOT SetSignalHigh AND
			NOT SetSignalLow AND
			NOT FlashSignal THEN

			SetOutPulse(IN:=TRUE,	PT:=DINT_TO_TIME(PulseTime)	);

			BitOutToSet:=SetOutPulse.Q;
			SetOutPulseActive:=TRUE;
			(* Pulse finished *)
			IF	NOT SetOutPulse.Q	THEN
				SetOutPulse(IN:=FALSE, PT:=T#0s);
				SetOutPulseActive:=FALSE;
			(* If no sensor check then state ok *)
			IF	NOT	InputAvailable OR
				(NOT CheckSignalHigh AND
				 NOT CheckSignalLow) THEN

				State:=STATE_OK;
				END_IF
			END_IF
		END_IF


		(* Set output with on and off time                         *)
		(*=========================================================*)
		IF	FlashSignal AND
			OnTime>0 AND
			OffTime>0 AND
			OutputAvailable AND

			NOT PulseOn AND
			NOT SetSignalHigh AND
			NOT SetSignalLow THEN

			TimerOn(IN:=TimerOff.Q = FALSE , PT:=DINT_TO_TIME(OnTime)); (* On time *)
			TimerOff(IN:=TimerOn.Q = TRUE, PT:=DINT_TO_TIME(OffTime));	(* Off time *)

			(* assign output *)
			IF 	NOT TimerOff.Q THEN
				BitOutToSet:=TRUE;
			ELSE
				BitOutToSet:=FALSE;
			END_IF

			(* If no sensor check then state ok *)
			IF 	NOT InputAvailable OR
				(NOT CheckSignalHigh AND
				 NOT CheckSignalLow) THEN

				State:=STATE_OK;
			END_IF
		
		
		END_IF
	
	
	(* Check input signal                                      *)
	(*=========================================================*)
	
		(* Check signal low and input is low*)
		IF	NOT 	BitInToCheck AND
			InputAvailable AND
			CheckSignalLow AND
			NOT CheckSignalHigh THEN

			(* Check input low and it is low *)
			TimerTimeOut(Start := FALSE, MTime := (sInit.MaxTime));
			State:=State_OK;

		(* Check input low and input is high*)
		ELSIF
			BitInToCheck AND
			InputAvailable AND
			CheckSignalLow AND
			NOT CheckSignalHigh THEN

			TimerTimeOut(Start := TRUE, MTime := (sInit.MaxTime));
			State:=STATE_ERROR (*INPUT_CHECKLOW*);
			FB_ReadXmlLineMsg.ID:='SensorFaultNotLow';

			TempErrorText:=sVisu.InstName;
			TempErrorText:=CONCAT(TempErrorText,' ');
			TempErrorText:=CONCAT(TempErrorText,sVisu.Description);
			TempErrorText:=CONCAT(TempErrorText,'  ');
			TempErrorText:=CONCAT(TempErrorText,FB_ReadXmlLineMsg.Text);

			Error.No:=1;

		(* Check input high *)
		ELSIF
			BitInToCheck AND
			InputAvailable AND
			NOT CheckSignalLow AND
			CheckSignalHigh THEN

			TimerTimeOut(Start := FALSE, MTime := (sInit.MaxTime));
			State:=State_OK;
	
		(* Check signal high and input is low*)
		ELSIF
			NOT BitInToCheck AND
			InputAvailable AND
			NOT CheckSignalLow AND
			CheckSignalHigh THEN

			TimerTimeOut(Start := TRUE, MTime := (sInit.MaxTime));
			State:=STATE_ERROR (*INPUT_CHECKHIGH*);
			FB_ReadXmlLineMsg.ID:='SensorFaultNotHigh';

			TempErrorText:=sVisu.InstName;
			TempErrorText:=CONCAT(TempErrorText,' :');
			TempErrorText:=CONCAT(TempErrorText,sVisu.Description);
			TempErrorText:=CONCAT(TempErrorText,'  ');
			TempErrorText:=CONCAT(TempErrorText,FB_ReadXmlLineMsg.Text);

			Error.No:=2;
		ELSE
			TimerTimeOut(Start := FALSE, MTime := (sInit.MaxTime));

			IF	SetSignalHigh AND
				CheckSignalLow AND
				NOT PulseOn AND
				NOT FlashSignal AND
				NOT CheckSignalHigh AND
				NOT CheckSignalLow THEN

				State:=STATE_WAIT;
			END_IF
		END_IF

		(* Timeout check high *)
		IF	TimerTimeOut.Timeout AND
			NOT ResetIntern AND
			State=INPUT_CHECKHIGH 	THEN

			State:=STATE_ERROR (*INPUT_CHECKHIGHFAULT*);
			FB_ReadXmlLineMsg.ID:='NotHhigh';

			TempErrorText:=sVisu.InstName;
			TempErrorText:=CONCAT(TempErrorText,' ');
			TempErrorText:=CONCAT(TempErrorText,sVisu.Description);
			TempErrorText:=CONCAT(TempErrorText,' ');
			TempErrorText:=CONCAT(TempErrorText,FB_ReadXmlLineMsg.Text);
			Error.No:=3;
		END_IF
		(* Timeout check low *)
		IF	TimerTimeOut.Timeout AND
			NOT ResetIntern AND
			State=INPUT_CHECKLOW THEN

			State:=STATE_ERROR (*INPUT_CHECKLOWFAULT*);
			FB_ReadXmlLineMsg.ID:='NotLow';

			TempErrorText:=sVisu.InstName;
			TempErrorText:=CONCAT(TempErrorText,' ');
			TempErrorText:=CONCAT(TempErrorText,sVisu.Description);
			TempErrorText:=CONCAT(TempErrorText,' ');
			TempErrorText:=CONCAT(TempErrorText,FB_ReadXmlLineMsg.Text);
			Error.No:=4;
		END_IF

	ELSE	(* No action *)
		(* Reset ok signal*)
		IF 	State = State_OK AND
			StateOK_CycleFlag THEN

			State:=STATE_WAIT;
		END_IF
	END_IF

END_IF	(* Init ok *)

(*--------------------------------------------------------------------
	Updating processtime (if State_RUN, STATE_ERROR, STATE_RESETS, or STATE_STOPPED)
--------------------------------------------------------------------*)
IF	( State=State_RUN OR
	State=STATE_ERROR OR
	State=STATE_RESETS OR
	State=STATE_STOPPED ) AND
	sInit.MaxTime<>0 AND
	InputAvailable<>0 THEN

	TimerTimeOut;
	ProcessTime:=TimerTimeOut.PTime;
END_IF

(*------------------------------------------------------------------
	Reset-Handling
  ------------------------------------------------------------------*)
ResetIntern:=Reset;

IF 	ResetIntern THEN

	TimerTimeOut (Start := FALSE, MTime := (sInit.MaxTime));
	State:= STATE_RESETS;
	BitOutToSet:=FALSE;
	SetOutPulse(IN:=FALSE);
	TimerOn(IN:=FALSE);
	TimerOff(IN:=FALSE);

	SetSignalHigh:=FALSE;		 		 	(* Signal set  HIGH *)
	SetSignalLow:=FALSE;		 			(* Signal set  LOW  *)
	PulseOn:=FALSE;		 			(* Signal pulse On *)
	FlashSignal:=FALSE;		 			(* Signal FLASH  *)
ELSE  (* IF Reset=FALSE *)
	IF 	State=STATE_RESETS THEN
		State:=STATE_WAIT;
	END_IF
END_IF

(*------------------------------------------------------------------
	Clear all input variables
  ------------------------------------------------------------------*)
Reset:= FALSE;
SetSignalLow:=FALSE;
SetSignalHigh:=FALSE;
PulseOn:=FALSE;
FlashSignal:=FALSE;
CheckSignalLow:= FALSE;
CheckSignalHigh:= FALSE;

(*------------------------------------------------------------------
	HomePosition
  ------------------------------------------------------------------*)
HomePositionInfo:=State_OK;

(* Check input signal *)
IF	sInit.HomePosSignal=0 AND
	BitInToCheck AND
	InputAvailable THEN
	HomePositionInfo:=11;
END_IF

IF	sInit.HomePosSignal=1 AND
	NOT BitInToCheck AND
	InputAvailable THEN
	HomePositionInfo:=10;
END_IF

(* Check output signal *)
IF	sInit.HomePosOutput=0 AND
	BitOutToSet AND
	OutputAvailable THEN
	HomePositionInfo:=21;
END_IF

IF	sInit.HomePosOutput=1 AND
	NOT BitOutToSet AND
	OutputAvailable THEN
	HomePositionInfo:=20;
END_IF


(* Generating home position*)
(* Zuweisung der Grundstellung*)
IF HomePositionInfo=State_OK THEN
	HomePosition:= TRUE;
ELSE
	HomePosition:= FALSE;
	ListHomeNOK(InstName:=sInit.InstName,Description:=FB_ReadXmlLineConf.Text);
END_IF

(* Objekt-Grundstellung verknüpfen mit GesamtGrundstellung *)
(* object-homeposition concat with mainhomeposition *)
gHomeOk:=gHomeOk AND HomePosition;

(*------------------------------------------------------------------
	Set Visu-Vars
  ------------------------------------------------------------------*)
sVisu.BitInName			:= sInit.BitInName;
sVisu.BitOutToSet		:= BitOutToSet;
sVisu.BitInToCheck		:= BitInToCheck;
sVisu.State				:= State;
sVisu.HomePosition		:= HomePosition;


(*Copy output-signal to output-var*)
SignalOut:=BitOutToSet;
(*Copy input-signal to output-var*)
SignalIn:=BitInToCheck;

(*------------------------------------------------------------------
	Error-Handling
  ------------------------------------------------------------------*)
ErrorElapsed(CLK:= Error.Text<>'');
IF ErrorElapsed.Q THEN
	Error.DateTime:=gVarDTSystemtime;
END_IF

IF Error.Text<>''	AND ST_Lng.b_EndChangeLng THEN
	Error.Typ:=0;

	(*Error.DateTime:=;*)
	ErrorHandler.AddError(
			ErrorToAdd:=Error,
			sVisu:=Visu.ErrorHandler);
END_IF

IF 	NOT Enable AND ModeSelect.Mode=MODE_MANUAL AND
	Error.Text='' AND
	strAnlayse<>'' THEN

	strAnlayse:=CONCAT(' +++ gesperrt durch : ',strAnlayse);

	LaufschriftAnalyse(
	N:= 40,
	StepWidth:=1,
	PT:= t#100ms ,
	Text:= strAnlayse,
	Display=>sVisu.ErrorString );

	strAnlayse:='';
ELSE
	IF Error.Text<>''	THEN
		TempString:=CONCAT(' --- ',Error.Text);
		LaufschriftObj(
		N:= 40,
		StepWidth:=1,
		PT:= t#100ms ,
		Text:= TempString,
		Display=>sVisu.ErrorString );
	ELSE
		sVisu.ErrorString:='';
	END_IF
END_IF

sVisu.InstName:=sInit.InstName;
sVisu.BitOutName:=sInit.BitOutName;
sVisu.BitInName:=sInit.BitInName;
sVisu.ErrorPresent:=Error.Text<>'';

FB_ReadXmlLineConf(
	Prefix:= 'CONFIG',
	ID:= sInit.InstName,
	File:= 'CONFIG.xml',
	Text=> sVisu.Description);

FB_ReadXmlLineMsg(
	Prefix:= 'MSG',
	ID:= ,
	File:= 'MSG.xml',
	Text=>);

IF 	State = STATE_ERROR THEN
	TempErrorText:=sInit.BitInName;
	TempErrorText:=CONCAT(TempErrorText,' :');
	TempErrorText:=CONCAT(TempErrorText,sVisu.Description);
	TempErrorText:=CONCAT(TempErrorText,' -> ');
	TempErrorText:=CONCAT(TempErrorText,FB_ReadXmlLineMsg.Text);
END_IF
END_FUNCTION_BLOCK

(* POU zLibrary/EpsonRobot/FB_EpsonRobot, ST *)
FUNCTION_BLOCK FB_EpsonRobot (*25.NOV 2010, Bernd Happach*)
VAR_INPUT
	ExecuteMove					: BOOL; 				(* Move to PositionNo *)
	PosNo							: DINT;					(* Position No from Robot *)
	PosOffset						: DINT;					(* Offset *)
	Override						: DINT;					(* Global override *)
	OffsetX							: REAL;					(* Offset X *)
	OffsetY							: REAL;					(* Offset Y *)
	OffsetZ							: REAL;					(* Offset Z *)
	ApplPara						: ARRAY[0..7] OF	REAL; (* Machinespecific Values *)

	SetToolOn						: BOOL;
	SetToolOff						: BOOL;

	Vel								: DINT;					(* Velocity for Linear Movements *)
	Acc								: DINT;					(* Acceleration 0..100% *)

	Enable							: BOOL; 				(* Enables the operations on the valve *)
	Reset							: BOOL; 				(* switch for resetting the object *)
	SFCCurrentStep					: STRING(80);			(* aktually step in the step flow chart *)
	SFCCurrentPOU					: STRING(80);			(* Name of the step flow chart *)
	sInit								: sEpsonRobotInit;		(* Initializingvalues to the Instance *)
	sToolSettings					: sEpsonRobotToolSettings;
	strAnlayse						: STRING(255);  		(*String to analyse Lockings*)

	CollisionActivated			:BOOL;
	Tool2Unit_AST						:BOOL;
END_VAR
VAR_OUTPUT
	State							: StateObject;			(* State of the object *)
	HomePosition					: BOOL;					(* object in home-position*)
	ActualPosition					: DINT;
	ActualArea						: DINT;
END_VAR
VAR_IN_OUT
	sVisu							: sEpsonRobotVisu;   	(* Structure for Visualisation *)
END_VAR
VAR
	RemOutStart					AT %Q* :	BOOL; 		(* Startbit für Task Main *)
	RemOutStop					AT %Q* :	BOOL; 		(* Task stoppen/ beenden *)
	RemOutPause					AT %Q* :	BOOL; 		(* Task anhalten *)
	RemOutCont					AT %Q* :	BOOL; 		(* Task fortsetzen *)
	RemOutReset					AT %Q* :	BOOL; 		(* Reset auf Roboter *)
	RemOutPowerOn				AT %Q* :	BOOL; 		(* Armleistung ein *)
	RemOutPowerOff				AT %Q* :	BOOL; 		(* Armleistung aus *)
	RemOutPowerHi					AT %Q* :	BOOL; 		(* Motor hohe Leistung ein *)
	RemOutSetToolOn				AT %Q* :	BOOL; 		(* Anforderung Ausgang Robotertool EIN *)
	RemOutSetToolOff				AT %Q* :	BOOL; 		(* Anforderung Ausgang Robotertool AUS *)

	RemInReady					AT %I* :	BOOL; 		(* Betriebsbereit von Roboter *)
	RemInRunning					AT %I* :	BOOL; 		(* Task (Main) aktiv von Roboter *)
	RemInPaused					AT %I* :	BOOL; 		(* Task angehalten - nicht abgebrochen! *)
	RemInError						AT %I* :	BOOL; 		(* quittierbare Störung von Roboter *)
	RemInEStopOn					AT %I* :	BOOL; 		(* Notaus-Kreis aktiv von Roboter *)
	RemInSafeguardOn				AT %I* :	BOOL; 		(* Schutzkreis (Türen) aktiv von Roboter *)
	RemInSError					AT %I* :	BOOL; 		(* nicht quittierbare Störung - Roboter AEG notwendig *)
	RemInWarning					AT %I* :	BOOL; 		(* Warnmeldung von Roboter *)
	RemInTcpIP_Wait				AT %I* :	BOOL; 		(* Handshake TcpIp-Verbindung *)
	RemInAreaBit1					AT %I* :	BOOL; 		(* Bereichsüberwachung Bit 1 *)
	RemInAreaBit2					AT %I* :	BOOL; 		(* Bereichsüberwachung Bit 2 *)
	RemInAreaBit4					AT %I* :	BOOL; 		(* Bereichsüberwachung Bit 4 *)

	RemInToolCoilA					AT %I* :  BOOL;		(* Rückmeldung Tool CoilA/ Ausgang 1 ist ein *)
	RemInToolCoilB					AT %I* :  BOOL;		(* Rückmeldung Tool CoilB/ Ausgang 2 ist ein *)
	RemInToolInitSensor				AT %I* :  BOOL;		(* Tool Ruhesensor *)
	RemInToolWorkSensor			AT %I* :  BOOL;		(* Tool Ruhesensor *)

	CollisionSensor					AT %I* :  BOOL;		(* Kollisonssensor Greifer*)

(* Internal used variables for movement Handling *)
	WorkingStep				: DINT;					(* Index for StateMachine *)
	PosNoLastMove				: DINT;					(* Position No from Robot *)
(* Init Handling *)
	InitStep						: INT;					(* Init Step StateMachine *)
	InitState						: BOOL :=	FALSE;		(* Internal State for initialising *)
	InitTimeOut					: TON;

	StepTimeOut				: TON;
(* Tool Handling *)
	ManToolOn					: TP;
	ManToolOff					: TP;

(* Error Handling *)
	TP_RemOutReset			: TP;

	TimerTimeOut				: CheckProcTime;	(* Timer generates timeout signal *)
	ProcessTime				: DINT;				(* Counts the time since starting operation *)

	Error						: ErrorStruct;
	ErrorElapsed				: R_TRIG;

	LaufschriftErrh				:FB_Laufschrift_STR255;
	LaufschriftObj				:FB_Laufschrift_STR255;
	LaufschriftAnalyse			:FB_Laufschrift_STR255;
	TempString					:STRING(255);

(* Internal used Variables tp send/receife data over TcpIP Socket *)
	ConnectionAlive				: BOOL;
	ConnectionTimer			: TON;
	TcpIP_Wait					: TON;
	ToolTimeOut				: TON;

	FP_Connected				: R_TRIG;


	DataIn						: sEpsonRobotRecvData;
	DataOut					: sEpsonRobotSendData;
	DataOutOld					: sEpsonRobotSendData;
	SendString					: STRING(255);

	ReceiveStep				: INT;

	FBClientServerConnection	: FB_ClientServerConnection;
	FBSocketReceive			: FB_SocketReceive;
	FBSocketSend				: FB_SocketSend;
	SocketHandle				: T_HSOCKET;

	_TON_SEND				: TP;

	eSocketState 				: E_SocketConnectionState;
	rxBuffer						: STRING(255);
	recString					: STRING(255);
	recBytes					: UDINT;

	StringWork					: STRING(255);
	ItemNo						: INT;
	StringStart					: INT;
	StringEnd					: INT;
	StringLen					: INT;
	ItemString					: STRING(255);
	ItemStringArray				: ARRAY [1..20] OF STRING;
	iPosArray					: INT;
(* Constants *)
	Delim						: STRING	:= ',';
	NoOfItems					: INT 		:= 16;


(* Visu Handling *)
	BtnMove					: VisuButton;
	BtnReset					: VisuButton;
	BtnPrgStart					: VisuButton;
	BtnPrgStop					: VisuButton;

	BtnToolOn					: VisuButton;
	BtnToolOff					: VisuButton;


	FB_ReadXmlLineConf		: FB_ReadXmlLine;
	FB_ReadXmlLineMsg		: FB_ReadXmlLine;

(*Kollisionsüberwachung*)
	fb_ton_collision				:TON;
	b_collision							: BOOL;
END_VAR
VAR CONSTANT
	RecBufferLen				: DINT := 100;
END_VAR
ToolTimeOut(IN:=,PT:=DINT_TO_TIME(sInit.ToolMaxTime));
Error.No:=0;
Error.Text:='';

Collision();
(*------------------------------------------------------------------
	Initialization
  ------------------------------------------------------------------*)
InitTimeOut(In:=NOT InitState,Pt:=T#5s);
IF 	NOT InitState THEN
	CASE InitStep OF
		0: (* Init Instance *)
			InitStep:=10;

		10:	InitStep:=50;
	
		50: (*Check IP-adress and Port*)
			InitStep:=100;

		100: (* Init Done *)
			IF	sInit.InstName <> '' THEN

				FOR iPosArray:=1 TO 20 DO
					(*Übersetzungen stehen in der CONFIG.xml*)
					sVisu.PosArray[iPosArray]:= '';
					sVisu.PosArray[iPosArray]:= CONCAT(	sVisu.PosArray[iPosArray],	sInit.InstName);
					sVisu.PosArray[iPosArray]:= CONCAT(	sVisu.PosArray[iPosArray],	'.PosArray[');
					sVisu.PosArray[iPosArray]:= CONCAT(	sVisu.PosArray[iPosArray],	INT_TO_STRING(iPosArray));
					sVisu.PosArray[iPosArray]:= CONCAT(	sVisu.PosArray[iPosArray],	']');
				END_FOR

			InitState:=TRUE;
			END_IF
	END_CASE

END_IF

IF InitState THEN
(*------------------------------------------------------------------
	Show and Read Visu Buttons
  ------------------------------------------------------------------*)
	BtnMove(	Button:=sVisu.BtnMove,
				Enable:=ModeSelect.Mode =	MODE_MANUAL AND
											Enable AND
											State=STATE_WAIT,
				TextOn:='Start'
							);

	BtnReset(	Button:=sVisu.BtnReset,
				Enable:=ModeSelect.Mode=MODE_MANUAL OR State=STATE_ERROR,
				TextOn:='Reset',
							);
	BtnPrgStart(	Button:=sVisu.BtnPrgStart,
				Enable:=ModeSelect.Mode=MODE_MANUAL ,
				TextOn:='Verbinden',
							);
	BtnPrgStop(	Button:=sVisu.BtnPrgStop,
				Enable:=ModeSelect.Mode=MODE_MANUAL ,
				TextOn:='Trennen',
							);
	BtnToolOn(	Button:=sVisu.BtnToolOn,
				Enable:=ModeSelect.Mode=MODE_MANUAL AND RemInRunning AND State=STATE_WAIT,
				TextOn:=sToolSettings.NameBtnToolOn,
							);
	BtnToolOff(	Button:=sVisu.BtnToolOff,
				Enable:=ModeSelect.Mode=MODE_MANUAL AND RemInRunning AND State=STATE_WAIT,
				TextOn:=sToolSettings.NameBtnToolOff,
							);
(*------------------------------------------------------------------
	EA-Handling
  ------------------------------------------------------------------*)
	ActualArea.0:=RemInAreaBit1;
	ActualArea.1:=RemInAreaBit2;
	ActualArea.2:=RemInAreaBit4;

	sVisu.ActualArea:=ActualArea;
(*------------------------------------------------------------------
	Manual Mode
  ------------------------------------------------------------------*)
	IF 	ModeSelect.Mode=MODE_MANUAL AND
		Enable THEN
		ExecuteMove:= BtnMove.Pressed;
		Reset:=Reset OR BtnReset.Pressed;
		IF 	ExecuteMove THEN
			(*Override:=10;*)
			PosNo:=sVisu.PosNo;
			OffsetX:=sVisu.OffsetX;
			OffsetY:=sVisu.OffsetY;
			OffsetZ:=sVisu.OffsetZ;
		END_IF

		ManToolOn(In:=BtnToolOn.Pressed,Pt:=T#1s);
		ManToolOff(In:=BtnToolOff.Pressed,Pt:=T#1s);
	END_IF

	RemOutPowerHi:=ModeSelect.Mode>MODE_MANUAL;
(*------------------------------------------------------------------
	Move-Handling
  ------------------------------------------------------------------*)
	TP_RemOutReset(In:=Reset,PT:=T#1s);

	RemOutReset:=	TP_RemOutReset.Q AND
					(	(	RemInError AND ( DataIn.ErrorCode < 8000 OR DataIn.ErrorCode > 8999 )	) OR
						RemInEStopOn OR
						RemInWarning OR
						RemInSError OR
						RemInSafeguardOn OR
						RemInPaused
						);
	RemOutPowerOff:=TP_RemOutReset.Q;
	RemOutCont:=TP_RemOutReset.Q;

	RemOutStart := 	(RemInReady AND
					NOT RemInRunning AND
					NOT RemInError AND
					NOT RemInEStopOn AND
					NOT RemInSafeguardOn AND
					NOT RemInSError AND
					NOT RemInWarning AND
					NOT TP_RemOutReset.Q AND
					vGlbImpuls_0500ms AND
					ModeSelect.Mode>MODE_MANUAL
					)	OR
					(RemInReady AND
					NOT RemInRunning AND
					NOT RemInError AND
					NOT RemInEStopOn AND
					NOT RemInSafeguardOn AND
					NOT RemInSError AND
					NOT RemInWarning AND
					NOT TP_RemOutReset.Q AND
					ModeSelect.Mode=MODE_MANUAL AND
					BtnPrgStart.Pressed
					);

	RemOutStop:= 	RemInRunning AND
					ModeSelect.Mode=MODE_MANUAL AND
					(BtnPrgStop.Pressed OR TP_RemOutReset.Q) OR
					RemInRunning AND
					ModeSelect.Mode>MODE_MANUAL AND
					TP_RemOutReset.Q;

	RemOutSetToolOn:=	(    ManToolOn.Q AND ModeSelect.Mode=MODE_MANUAL ) OR
						(    SetToolOn  AND ModeSelect.Mode>MODE_MANUAL );

	RemOutSetToolOff:=	 (  ManToolOff.Q AND ModeSelect.Mode=MODE_MANUAL ) OR
						 (  SetToolOff AND ModeSelect.Mode>MODE_MANUAL );

(* Generate Flags To Start Movement *)

	CASE WorkingStep OF
	0: (* State STATE_WAIT *)

		State:=STATE_WAIT;

		IF 	ExecuteMove THEN
			WorkingStep:=10;
			(* Start Execution Time *)
			TimerTimeOut.Start:=TRUE;
			State:=STATE_RUN;
		END_IF
	10: (* Check Star Conditions *)
		IF  ConnectionAlive AND
			RemInRunning THEN
			WorkingStep:=100;
		ELSE
			State:=STATE_ERROR;
		END_IF
	100:(* Handle Robot EA´s if nessecary *)
			StepTimeOut(In:=FALSE);
			WorkingStep:=200;
	200:(* Start Movement - Assign Variables *)

			PosNoLastMove:=PosNo + PosOffset;

			DataOut.TelNo:=2;
			DataOut.PosNo:=PosNo + PosOffset;
			DataOut.Override:=Override;
			DataOut.OffsetX:=OffsetX;
			DataOut.OffsetY:=OffsetY;
			DataOut.OffsetZ:=OffsetZ;
			DataOut.ApplPara:=ApplPara;
			DataOut.Vel:=Vel;
			DataOut.Acc:=Acc;

			StepTimeOut(In:=DataIn.TelNo<>0 AND DataIn.TelNo<>DataOut.TelNo,Pt:=DINT_TO_TIME(sInit.MaxTime));
			IF 	DataIn.TelNo=DataOut.TelNo THEN
				WorkingStep:=201;
				ActualPosition:=0;

			ELSIF StepTimeOut.Q THEN
				(* Error *)
				State:=STATE_ERROR;
				FB_ReadXmlLineMsg.ID:='StartError';
				Error.No:=1;
				Error.Text:=sInit.InstName;
				Error.Text:=CONCAT(Error.Text,': ');
				Error.Text:=CONCAT(Error.Text,sInit.Description);
				Error.Text:=CONCAT(Error.Text,' - ');
				Error.Text:=CONCAT(Error.Text,FB_ReadXmlLineMsg.Text);
				WorkingStep:=999;
			END_IF

	201:(* Dummy step *)
			StepTimeOut(In:=FALSE);
			WorkingStep:=210;

	210:(* Wait Movement Done *)
			StepTimeOut(In:=DataIn.PosNo <>0 AND DataIn.PosNo<>DataOut.PosNo,Pt:=DINT_TO_TIME(sInit.MaxTime));
			IF 	DataIn.PosNo=DataOut.PosNo THEN
				DataOut.TelNo:=0;
				DataOut.PosNo:=0;
				ActualPosition:=DataIn.PosNo;
				WorkingStep:=220;
			ELSIF
				StepTimeOut.Q THEN
				(* Error *)
				State:=STATE_ERROR;
				FB_ReadXmlLineMsg.ID:='PosNoNotDefined';
				Error.No:=1;
				Error.Text:=sInit.InstName;
				Error.Text:=CONCAT(Error.Text,': ');
				Error.Text:=CONCAT(Error.Text,sInit.Description);
				Error.Text:=CONCAT(Error.Text,' - ');
				Error.Text:=CONCAT(Error.Text,FB_ReadXmlLineMsg.Text);
				WorkingStep:=999;
			END_IF
	220:(* Quit Telegramm Done *)
			IF 	DataIn.PosNo=0 AND DataIn.TelNo=0 THEN
				IF 	SetToolOn AND sInit.WithToolHandling THEN
					WorkingStep:=300;
				ELSIF
					SetToolOff AND sInit.WithToolHandling THEN
					WorkingStep:=400;
				ELSE
					WorkingStep:=1000;
				END_IF
			END_IF
	300: (* Check tool in workposition *)
			IF sToolSettings.NameWorkSensor<>'xxxx' THEN
				ToolTimeOut.IN:=TRUE;
				IF 	RemInToolWorkSensor THEN
					WorkingStep:=1000;
				ELSIF
					ToolTimeOut.Q THEN
					State:=STATE_ERROR;
					FB_ReadXmlLineMsg.ID:='TimeoutToolWork';
					Error.No:=1;
					Error.Text:=sInit.InstName;
					Error.Text:=CONCAT(Error.Text,': ');
					Error.Text:=CONCAT(Error.Text,sInit.Description);
					Error.Text:=CONCAT(Error.Text,' - ');
					Error.Text:=CONCAT(Error.Text,FB_ReadXmlLineMsg.Text);
				END_IF
			ELSE
				WorkingStep:=1000;
			END_IF

	400: (* Check tool in initposition *)
			IF 	sToolSettings.NameInitSensor<>'xxxx' THEN
				ToolTimeOut.IN:=TRUE;
				IF 	RemInToolInitSensor THEN
					WorkingStep:=1000;
				ELSIF
					ToolTimeOut.Q THEN
					State:=STATE_ERROR;
					FB_ReadXmlLineMsg.ID:='TimeoutToolInit';
					Error.No:=1;
					Error.Text:=sInit.InstName;
					Error.Text:=CONCAT(Error.Text,': ');
					Error.Text:=CONCAT(Error.Text,sInit.Description);
					Error.Text:=CONCAT(Error.Text,' - ');
					Error.Text:=CONCAT(Error.Text,FB_ReadXmlLineMsg.Text);	
				END_IF
			ELSE
				WorkingStep:=1000;
			END_IF

	999: (* State Error *)
			State:=STATE_ERROR;
			StepTimeOut(In:=FALSE);
			TimerTimeOut.Start:=FALSE;
	1000: (* State OK *)
			State:=STATE_OK;
			TimerTimeOut.Start:=FALSE;
			ToolTimeOut.IN:=FALSE;
			IF 	NOT ExecuteMove THEN (*OR PosNoLastMove<>PosNo*)
				WorkingStep:=0;
				State:=STATE_WAIT;
				ProcessTime:=TimerTimeOut.PTime;
			END_IF
	END_CASE

(*--------------------------------------------------------------------
		Handle Timeout
  --------------------------------------------------------------------*)
	IF 	TimerTimeOut.Timeout AND
		State<>STATE_ERROR THEN

		State:=STATE_TIMEOUT;
		Error.No:=1;
		Error.Text:=sInit.InstName;
		Error.Text:=CONCAT(Error.Text,': ');
		Error.Text:=CONCAT(Error.Text,sInit.Description);
		Error.Text:=CONCAT(Error.Text,' - ');
		Error.Text:=CONCAT(Error.Text,' [Rob. Error code: ');
		Error.Text:=CONCAT(Error.Text,DINT_TO_STRING(DataIn.ErrorCode));
		Error.Text:=CONCAT(Error.Text,']');

		FB_ReadXmlLineMsg.ID:=DINT_TO_STRING(DataIn.ErrorCode);

		CASE DataIn.ErrorCode OF
			8000:
				Error.Text:=CONCAT(Error.Text,FB_ReadXmlLineMsg.Text);
			8001:
				Error.Text:=CONCAT(Error.Text,FB_ReadXmlLineMsg.Text);
			8002:
				Error.Text:=CONCAT(Error.Text,FB_ReadXmlLineMsg.Text);
			8003:
				Error.Text:=CONCAT(Error.Text,FB_ReadXmlLineMsg.Text);
			8006:
				Error.Text:=CONCAT(Error.Text,FB_ReadXmlLineMsg.Text);
			8010:
				Error.Text:=CONCAT(Error.Text,FB_ReadXmlLineMsg.Text);
			8011:
				Error.Text:=CONCAT(Error.Text,FB_ReadXmlLineMsg.Text);
			8012:
				Error.Text:=CONCAT(Error.Text,FB_ReadXmlLineMsg.Text);
			8013:
				Error.Text:=CONCAT(Error.Text,FB_ReadXmlLineMsg.Text);
			8014:
				Error.Text:=CONCAT(Error.Text,FB_ReadXmlLineMsg.Text);
			8015:
				Error.Text:=CONCAT(Error.Text,FB_ReadXmlLineMsg.Text);
			8016:
				Error.Text:=CONCAT(Error.Text,FB_ReadXmlLineMsg.Text);
		END_CASE
	END_IF

(*--------------------------------------------------------------------
		Call Timers
  --------------------------------------------------------------------*)
	TimerTimeOut(MTime:=sInit.MaxTime);

(*--------------------------------------------------------------------
		Updating processtime (if State_RUN, STATE_TIMEOUT, STATE_RESETS, or STATE_STOPPED)
  --------------------------------------------------------------------*)
	IF	(State=STATE_OK OR
		State=STATE_TIMEOUT OR
		State=STATE_RESETS OR
		State=STATE_STOPPED) AND
		 sInit.MaxTime<>0 THEN
		ProcessTime:=TimerTimeOut.PTime;
	END_IF

(*--------------------------------------------------------------------
	HomePosition
  --------------------------------------------------------------------*)
	IF 	(ActualPosition MOD 1000)=1 AND ConnectionAlive THEN
		HomePosition:=TRUE;
	ELSE
		HomePosition:=FALSE;
	END_IF

	(* Generating home position*)
	IF NOT HomePosition THEN
		ListHomeNOK(InstName:=sInit.InstName,Description:=FB_ReadXmlLineConf.Text);
	END_IF

	(* Object-homeposition concat with mainhomeposition *)
	gHomeOk:=gHomeOk AND HomePosition;

(*------------------------------------------------------------------
	Update Visu
  ------------------------------------------------------------------*)
	sVisu.InstName:=sInit.InstName;
	sVisu.Description:=sInit.Description;
	sVisu.TcpIpAdress:=sInit.TcpIPAdress;
	CASE eSocketState OF
		eSOCKET_CONNECTED: sVisu.SocketState:='Connected';
		eSOCKET_DISCONNECTED: sVisu.SocketState:='Disconnected';
		eSOCKET_SUSPENDED: sVisu.SocketState:='Suspended';
	END_CASE
	sVisu.State:=State;

	sVisu.ProcessTime:=ProcessTime;
	sVisu.HomePosition:=HomePosition;
	sVisu.ActualPosition:=ActualPosition;
	sVisu.ConnectionAlive:=ConnectionAlive;

	sVisu.PosX:=DataIn.PosX;
	sVisu.PosY:=DataIn.PosY;
	sVisu.PosZ:=DataIn.PosZ;

	sVisu.PosOffset:= 			PosOffset;

(* EA's from Robot *)
	sVisu.RemOutStart:=			RemOutStart; 		(* For Moving to WorkPosition *)
	sVisu.RemOutStop:=			RemOutStop; 		(* For Moving to WorkPosition *)
	sVisu.RemOutPause	:= 		RemOutPause; 		(* For Moving to WorkPosition *)
	sVisu.RemOutCont:=			RemOutCont; 		(* For Moving to WorkPosition *)
	sVisu.RemOutReset:=		RemOutReset; 		(* For Moving to WorkPosition *)
	sVisu.RemOutPowerOn:=	RemOutPowerOn; 		(* For Moving to WorkPosition *)
	sVisu.RemOutPowerOff:=	RemOutPowerOff; 		(* For Moving to WorkPosition *)
	sVisu.RemOutPowerHi:=		RemOutPowerHi; 		(* For Moving to WorkPosition *)

	sVisu.RemInReady:=			RemInReady; 		(* For Moving to WorkPosition *)
	sVisu.RemInRunning	:=		RemInRunning; 		(* For Moving to WorkPosition *)
	sVisu.RemInPaused:=		RemInPaused; 		(* For Moving to WorkPosition *)
	sVisu.RemInError:=			RemInError; 		(* For Moving to WorkPosition *)
	sVisu.RemInEStopOn:=		RemInEStopOn; 		(* For Moving to WorkPosition *)
	sVisu.RemInSafeguardOn:=	RemInSafeguardOn; 		(* For Moving to WorkPosition *)
	sVisu.RemInSError:=			RemInSError; 		(* For Moving to WorkPosition *)
	sVisu.RemInWarning	:=		RemInWarning; 		(* For Moving to WorkPosition *)

	sVisu.RemInTcpIP_Wait	:=	RemInTcpIP_Wait; 		(* For Moving to WorkPosition *)
	sVisu.RemInAreaBit1	:=		RemInAreaBit1; 		(* For Moving to WorkPosition *)
	sVisu.RemInAreaBit2	:=		RemInAreaBit2; 		(* For Moving to WorkPosition *)
	sVisu.RemInAreaBit4	:=		RemInAreaBit4; 		(* For Moving to WorkPosition *)

	sVisu.WithToolHandling:=		sInit.WithToolHandling;
	sVisu.NameCoilA:=				sToolSettings.NameCoilA;
	sVisu.NameCoilB:=				sToolSettings.NameCoilB;
	sVisu.NameInitSensor:=			sToolSettings.NameInitSensor;
	sVisu.NameWorkSensor:=		sToolSettings.NameWorkSensor;
	sVisu.RemInToolCoilA:=			RemInToolCoilA;
	sVisu.RemInToolCoilB:=			RemInToolCoilB;
	sVisu.RemInToolInitSensor:=		RemInToolInitSensor;
	sVisu.RemInToolWorkSensor	:=	RemInToolWorkSensor;
	sVisu.RemOutSetToolOn	:=		RemOutSetToolOn;
	sVisu.RemOutSetToolOff	:=		RemOutSetToolOff;

(*------------------------------------------------------------------
	Check ConnectionState
  ------------------------------------------------------------------*)
(* Toggle Alive Bit *)

	ConnectionTimer(IN:=DataOut.Alive<>DataIn.Alive OR eSocketState<>eSOCKET_CONNECTED , PT:= t#2000ms );
	ConnectionAlive:=NOT ConnectionTimer.Q;
	
	IF 	DataOut.Alive=DataIn.Alive OR
		(NOT ConnectionAlive AND eSocketState=eSOCKET_CONNECTED AND vGlbImpuls_1000ms) THEN
		IF DataOut.Alive=0 THEN
			DataOut.Alive:=1;
		ELSE
			DataOut.Alive:=0;
		END_IF
	END_IF

	IF 	eSocketState<>eSOCKET_CONNECTED THEN
		DataOut.Alive:=0;
	END_IF
(* Create Sendstring *)


	sendString:=CONCAT(DINT_TO_STRING(DataOut.Alive),Delim);
	sendString:=CONCAT(sendString,DINT_TO_STRING(DataOut.TelNo));
	sendString:=CONCAT(sendString,Delim);
	sendString:=CONCAT(sendString,DINT_TO_STRING(DataOut.PosNo));
	sendString:=CONCAT(sendString,Delim);
	sendString:=CONCAT(sendString,DINT_TO_STRING(DataOut.Override));
	sendString:=CONCAT(sendString,Delim);
	sendString:=CONCAT(sendString,DINT_TO_STRING(DataOut.Vel));
	sendString:=CONCAT(sendString,Delim);
	sendString:=CONCAT(sendString,DINT_TO_STRING(DataOut.Acc));
	sendString:=CONCAT(sendString,Delim);
	sendString:=CONCAT(sendString,REAL_TO_STRING(DataOut.OffsetX * 1000.0));
	sendString:=CONCAT(sendString,Delim);
	sendString:=CONCAT(sendString,REAL_TO_STRING(DataOut.OffsetY * 1000.0));
	sendString:=CONCAT(sendString,Delim);
	sendString:=CONCAT(sendString,REAL_TO_STRING(DataOut.OffsetZ * 1000.0));
	sendString:=CONCAT(sendString,Delim);
	sendString:=CONCAT(sendString,REAL_TO_STRING(DataOut.ApplPara[0] * 1000.0));
	sendString:=CONCAT(sendString,Delim);
	sendString:=CONCAT(sendString,REAL_TO_STRING(DataOut.ApplPara[1] * 1000.0));
	sendString:=CONCAT(sendString,Delim);
	sendString:=CONCAT(sendString,REAL_TO_STRING(DataOut.ApplPara[2] * 1000.0));
	sendString:=CONCAT(sendString,Delim);
	sendString:=CONCAT(sendString,REAL_TO_STRING(DataOut.ApplPara[3] * 1000.0));
	sendString:=CONCAT(sendString,Delim);
	sendString:=CONCAT(sendString,REAL_TO_STRING(DataOut.ApplPara[4] * 1000.0));
	sendString:=CONCAT(sendString,Delim);
	sendString:=CONCAT(sendString,REAL_TO_STRING(DataOut.ApplPara[5] * 1000.0));
	sendString:=CONCAT(sendString,Delim);
	sendString:=CONCAT(sendString,REAL_TO_STRING(DataOut.ApplPara[6] * 1000.0));
	sendString:=CONCAT(sendString,Delim);
	sendString:=CONCAT(sendString,REAL_TO_STRING(DataOut.ApplPara[7] * 1000.0));
	sendString:=CONCAT(sendString,Delim);

	FP_Connected(CLK:= eSocketState=eSOCKET_CONNECTED);

	IF 	(MEMCMP(ADR(DataOut),ADR(DataOutOld),SIZEOF(DataOut))<>0 AND eSocketState=eSOCKET_CONNECTED) OR FP_Connected.Q THEN
		FBSocketSend.bExecute:=TRUE;
		DataOutOld:=DataOut;
	END_IF

	TcpIP_Wait(IN:=RemInTcpIP_Wait , PT:=t#5ms );

	CASE ReceiveStep OF
	0: (* Waiting for Robot is Ready to Connect *)
		IF 	TcpIP_Wait.Q THEN
			ReceiveStep:=1;
		END_IF
	1: (* Connect *)
		FBClientServerConnection.bEnable:= TRUE;
		IF 	FBClientServerConnection.bBusy THEN
			ReceiveStep:=2;
		END_IF
	2:(* Connected *)
		IF 	eSocketState=eSOCKET_CONNECTED THEN
			ReceiveStep:=10;
		END_IF
	10:
		IF 	SocketHandle.handle>0 THEN
			ReceiveStep:=11;
		END_IF
	11:(* Start to Receive *)
		rxBuffer:='';
	 	FBSocketReceive.bExecute:=TRUE;
		IF 	FBSocketReceive.bBusy THEN
			ReceiveStep:=12;
		END_IF
	12:(* Rec Done *)
		FBSocketReceive.bExecute:=TRUE;
		IF 	NOT FBSocketReceive.bBusy AND NOT
			FBSocketReceive.bError AND
			FBSocketReceive.nRecBytes>99 THEN
			(* Data Received *)
			ReceiveStep:=20;
		ELSIF
			NOT FBSocketReceive.bBusy AND NOT
			FBSocketReceive.bError AND
			FBSocketReceive.nRecBytes=0 THEN
			(* NO Data Received *)
			ReceiveStep:=10;
		ELSIF
			NOT FBSocketReceive.bBusy AND NOT
			FBSocketReceive.bError AND
			FBSocketReceive.nRecBytes>0 THEN
			(* NO Data Received *)
			ReceiveStep:=10;

		ELSIF
			NOT FBSocketReceive.bBusy AND
			FBSocketReceive.bError THEN
			(* ERROR *)
			ReceiveStep:=100;
		END_IF
	20:(* Decrypt Data *)
		recString:=rxBuffer;
	  (* Handle String *)
		StringWork:=recString;
		FOR ItemNo:=1 TO NoOfItems DO
			StringStart:=1;
			StringEnd:=FIND(StringWork, Delim);
			IF 	StringEnd<>0 THEN
				StringLen:=StringEnd-StringStart;
				ItemString:=MID(StringWork,StringLen,StringStart);
				StringWork:=REPLACE(StringWork,'',StringLen+1,StringStart);
				ItemStringArray[ItemNo]:=ItemString;
			ELSE
				(* Delete $r and $n *)
				IF 	StringWork<>'' THEN
					StringStart:=FIND(StringWork, '$R');
					IF 	StringStart <> 0 THEN
						StringLen:=LEN(StringWork)-(StringStart-1);
						StringWork:=REPLACE(StringWork,'',StringLen,StringStart);
					END_IF

					StringStart:=FIND(StringWork, 'X');
					IF 	StringStart <> 0 THEN
						StringLen:=LEN(StringWork)-(StringStart-1);
						StringWork:=REPLACE(StringWork,'',StringLen,StringStart);
					END_IF

					StringStart:=FIND(StringWork, '$N');
					IF 	StringStart <> 0 THEN
						StringLen:=LEN(StringWork)-(StringStart-1);
						StringWork:=REPLACE(StringWork,'',StringLen,StringStart);
					END_IF

					ItemStringArray[ItemNo]:=StringWork;
				END_IF
				EXIT;
			END_IF
		END_FOR (* ItemNo *)

		ReceiveStep:=22;
	22: (*Check Data*)
		IF 	ItemStringArray[1]='BEG' THEN
			DataIn.Alive:=STRING_TO_DINT(ItemStringArray[2]);
			DataIn.TelNo:=STRING_TO_DINT(ItemStringArray[3]);
			DataIn.PosNo:=STRING_TO_DINT(ItemStringArray[4]);
			DataIn.PosX:=STRING_TO_REAL(ItemStringArray[5]) / 1000.0;
			DataIn.PosY:=STRING_TO_REAL(ItemStringArray[6]) / 1000.0;
			DataIn.PosZ:=STRING_TO_REAL(ItemStringArray[7]) / 1000.0;

			DataIn.ApplPara[0]:=STRING_TO_REAL(ItemStringArray[8]) / 1000.0;
			DataIn.ApplPara[1]:=STRING_TO_REAL(ItemStringArray[9]) / 1000.0;
			DataIn.ApplPara[2]:=STRING_TO_REAL(ItemStringArray[10]) / 1000.0;
			DataIn.ApplPara[3]:=STRING_TO_REAL(ItemStringArray[11]) / 1000.0;
			DataIn.ApplPara[4]:=STRING_TO_REAL(ItemStringArray[12]) / 1000.0;
			DataIn.ApplPara[5]:=STRING_TO_REAL(ItemStringArray[13]) / 1000.0;
			DataIn.ApplPara[6]:=STRING_TO_REAL(ItemStringArray[14]) / 1000.0;
			DataIn.ApplPara[7]:=STRING_TO_REAL(ItemStringArray[15]) / 1000.0;
			DataIn.ErrorCode	:=STRING_TO_DINT(ItemStringArray[16]);
			ReceiveStep:=10;
		ELSE
			ReceiveStep:=10;
		END_IF
	100: (* Errorhandler -> Reconnect *)
		FBClientServerConnection.bEnable:= FALSE;
		ReceiveStep:=101;

	101:
		IF	eSocketState=eSOCKET_DISCONNECTED THEN
			ReceiveStep:=0;
		END_IF
	END_CASE

	FBClientServerConnection(
		sSrvNetID:=	'',
		nMode:= CONNECT_MODE_ENABLEDBG,
		sRemoteHost:= sInit.TcpIPAdress,
		nRemotePort:= sInit.TcpIPSocket,
		tReconnect:= t#10s,
		hSocket=> SocketHandle,
		eState=> eSocketState);


	FBSocketReceive(
		sSrvNetId:= '',
		hSocket:= SocketHandle,
		cbLen:= RecBufferLen,
		pDest:= ADR(rxBuffer),
		tTimeout:= t#1s,
		nRecBytes=> recBytes);

	FBSocketReceive.bExecute:=FALSE;
	_TON_SEND(IN:=FBSocketSend.bExecute , PT:=t#10ms );
	FBSocketSend(
		sSrvNetId:= '',
		hSocket:= SocketHandle,
		cbLen:= LEN(sendString),
		pSrc:= ADR(sendString),
		tTimeout:= t#1s
	 );

	FBSocketSend.bExecute:=FALSE;

END_IF (* Init OK *)

(*------------------------------------------------------------------
	Reset-Handling
  ------------------------------------------------------------------*)
IF 	Reset THEN
	RemOutStart:=FALSE;
	RemOutStop:=TRUE;
	RemOutReset:=TRUE;
	State:=STATE_RESETS;
	WorkingStep:=0;
	ProcessTime:=0;
	TimerTimeOut.Start:=FALSE;
	DataOut.TelNo:=0;
	DataOut.PosNo:=0;
	DataOut.Alive:=0;
	b_collision:=FALSE;
	IF	NOT ConnectionAlive THEN
		ReceiveStep:=100;
	END_IF
END_IF


(*------------------------------------------------------------------
	Error-Handling
  ------------------------------------------------------------------*)
ErrorElapsed(CLK:= Error.Text<>'');
IF 	ErrorElapsed.Q THEN
	Error.DateTime:=gVarDTSystemtime;
END_IF

IF 	Error.Text<>'' AND
	ST_Lng.b_EndChangeLng THEN
	Error.Typ:=0;

	(*Error.DateTime:=;*)
	ErrorHandler.AddError(	ErrorToAdd:=Error,
							sVisu:=Visu.ErrorHandler);

END_IF

IF 	NOT Enable AND
	ModeSelect.Mode=MODE_MANUAL AND
	Error.Text='' AND
	strAnlayse<>'' THEN

	strAnlayse:=CONCAT(' +++ gesperrt durch : ',strAnlayse);

	LaufschriftAnalyse(
	N:= 40,
	StepWidth:=1,
	PT:= t#100ms ,
	Text:= strAnlayse,
	Display=>sVisu.ErrorString );

	strAnlayse:='';
ELSE
	IF 	Error.Text<>'' THEN
		TempString:=CONCAT(' --- ',Error.Text);
		LaufschriftObj(
		N:= 80,
		StepWidth:=1,
		PT:= t#100ms ,
		Text:= TempString,
		Display=>sVisu.ErrorString );
	ELSE
		sVisu.ErrorString:='';
	END_IF
END_IF
sVisu.ErrorPresent:=sVisu.ErrorString='';
(*------------------------------------------------------------------
	Reset Inputs
  ------------------------------------------------------------------*)

IF 	state=STATE_WAIT OR
	state=STATE_RESETS OR
	state=STATE_OK THEN
	ExecuteMove:=FALSE;
	PosNo:=0;
	Enable:=FALSE;
	Reset:= FALSE;
	SetToolOn:= FALSE;
	SetToolOff:= FALSE;

	(*Override:=	0;			(* Global override *)*)
	OffsetX	:=	0.0;			(* Offset X *)
	OffsetY	:=	0.0;			(* Offset Y *)
	OffsetZ	:=	0.0;			(* Offset Z *)
	ApplPara[0]:=0.0; 		(* Machinespecific Values *)
	ApplPara[1]:=0.0; 		(* Machinespecific Values *)
	ApplPara[2]:=0.0; 		(* Machinespecific Values *)
	ApplPara[3]:=0.0; 		(* Machinespecific Values *)
	ApplPara[4]:=0.0; 		(* Machinespecific Values *)
	ApplPara[5]:=0.0; 		(* Machinespecific Values *)
	ApplPara[6]:=0.0; 		(* Machinespecific Values *)
	ApplPara[7]:=0.0; 		(* Machinespecific Values *)

END_IF


sVisu.BitName:=sInit.BitName;
sVisu.InstName:=sInit.InstName;

FB_ReadXmlLineConf(
	Prefix:= 'CONFIG',
	ID:= sInit.InstName,
	File:= 'CONFIG.xml',
	Text=> sVisu.Description );

FB_ReadXmlLineMsg(
	Prefix:= 'MSG',
	ID:= ,
	File:= 'MSG.xml',
	Text=>);
END_FUNCTION_BLOCK
ACTION Collision:
fb_ton_collision(IN:=collisionSensor AND Tool2Unit_AST AND ActualArea = 6,PT:= t#100ms, Q=> , ET=> );
IF 	fb_ton_collision.Q THEN
	b_collision:= TRUE;
END_IF

IF CollisionActivated THEN
	IF 	b_collision THEN
		RemOutStart:=FALSE;
		RemOutStop:=TRUE;
		WorkingStep:=0;
		State:=STATE_ERROR;
		Error.Text:=CONCAT('Error movement: ','collision');
		Error.No:=1;
	END_IF
END_IF
END_ACTION

(* POU zLibrary/ept/Achse/fb_72x1_Achse, ST *)
FUNCTION_BLOCK fb_72x1_Achse   (*Coe-Online 7010.03 (CSV) velocity mode*)
VAR_INPUT
	Stop				:BOOL;			(*aktiven Verfahrbefehl beenden*)
	Reset				:BOOL;			(*Fehler quttieren*)
	MotorOn				:BOOL;			(*Regelung einschalten*)
	MotorOff			:BOOL;			(*Regelung abschalten*)
	NotausOK			:BOOL;
	Override			:DINT;
	Offset				:REAL;			(*  *)
	Vorgabe_Velo		:DINT;			(*in U/min oder mm/min*)
	MoveAbs				:BOOL;			(*startet Positionierung absolut*)
	MoveRel				:BOOL;			(*startet Positionierung relativ*)
	Vorgabe_Pos_Abs		:LREAL:=0;		(*auf diese Position wird bei start MoveAbs gefahren (mm oder Grad)*)
	Vorgabe_Pos_Rel		:LREAL:=0;		(*um diesen Wert wird die Achse bei start MoveRel gefahren (mm oder Grad)*)
	MoveP				:BOOL;			(*Achse bewegt sich in positiver Richtung solange MoveP TRUE ist, oder bis zum Softwarelimit*)
	MoveN				:BOOL;			(*Achse bewegt sich in negativer Richtung solange MoveN TRUE ist, oder bis zum Softwarelimit*)
	bMove				:BOOL;
	sConfig				:st_config_axis;	(*Initialisierung der Achse*)
	sPosList			:ARRAY [1..NO_OF_POS_AXIS] OF st_Pos;

	e_Position			AT %I* :UDINT;
	e_Statusword		AT %I* :UINT;
	e_Velocity			AT %I* :DINT;
	e_Torque			AT %I* :INT;
	e_Following_Error	AT %I* :DINT; 	(*Schleppfehler*)
	e_Toggle			AT %I* :BOOL;
	e_State				AT %I* :UINT;

END_VAR
VAR_OUTPUT
	a_Controlword		AT %Q* :UINT;
	a_Target_Velocity	AT %Q*: DINT;
	a_Target_Position	AT %Q* :UDINT;
	Torque				:ARRAY [1..NO_OF_Torque] OF INT;

	Busy				:BOOL;
	Done				:BOOL;		(*Achse steht auf Position*)
	Error_				:BOOL;
	Ready				:BOOL;
	On					:BOOL;		(*Motor in Regelung*)
	On_Position			:BOOL;		(*Achse steht auf Position*)
	Connect				:BOOL;		(*KLemme ist mit PLC verbunden*)
END_VAR
VAR_IN_OUT
	sVisu				:sDigInVisu;
END_VAR
VAR
	sHelp				:st_Help_axis;
	fb_state_entry		:ST_StateEntry;

	sFb					:st_fb_axis;

	sSm					:st_sm_axis;		(*Störmeldungen*)
	sSmEmpty			:st_sm_axis;
	sCtrl				:st_ctrl_Axis;		(*Control und Status*)
	sCtrlEmpty			:st_ctrl_Axis;

	sVisuAxis			:st_Visu_axis;		(*Taster der Visu*)
	sSdo				:st_sdo;

	(*Variablen für Behr Meldungen*)
	TempErrorText		:STRING(255);
	ProcessTime			:DINT;				(* Counts the time in steps of 100ms since starting operation *)
	Error				:ErrorStruct;
	LaufschriftErrh		:FB_Laufschrift;
	LaufschriftObj		:FB_Laufschrift;

	(*Regler*)
	sVelo				:st_Velo_axis;		(*Geschwindigkeiten*)
	sRegler				:st_PID_axis;		(*Var zur ermittling der Ausgabegeschwindigkeit*)
	sPos				:st_Pos_axis;		(*Positionen*)

	FB_ReadXmlLineConf	:FB_ReadXmlLine;
	FB_ReadXmlLineMsg	:FB_ReadXmlLine;

END_VAR
VAR_TEMP
	i					:INT;
END_VAR

VAR CONSTANT
	NO_OF_Torque		: INT :=50;
END_VAR
(*======================================================
   FB: fb_72x1_Achse (Achse ohne NC verfahren)
 ------------------------------------------------------
   Auth: 		Werner Friedl    						 
   Date: 		18.04.2018   						     
   Rev.: 		1.0	
   Desc:		siehe Aktion " Description "
 ========================================================*)
sub_connect();
sub_Visu();
IF 	NOT sHelp.b_init AND
	sConfig.Aktiv AND
	e_Position<> 0 AND
	Connect  THEN
	sHelp.b_init:=TRUE;
	sPos.r_18bit:=EXPT(2,18);		(*262144 für e_Velocity *)
	sPos.r_20bit:=EXPT(2,20);		(*1048576 für e_Position*)
	sPos.r_32bit:=EXPT(2,32);		(*4294967295 für Überlauf*)
	sConfig.UeberlaufControl_on:=sConfig.SW_Limit_on;
END_IF

IF	sConfig.Aktiv AND
	sConfig.Skalierfaktor <> 0 AND
	sConfig.Getriebefaktor <>0  AND
	sHelp.b_init AND
	Connect THEN
	sub_Regler();
	sub_Pos();
	sub_rec_Torque();
END_IF

Btn_init();
sub_ctrl();
sub_sdo();
sub_fb();

(* Toplevel *)
IF 	fb_state_entry.i16_next_step > INIT AND fb_state_entry.i16_next_step < FEHLER THEN
	IF 	sFb.ton_uez.Q AND NOT sCtrl.in.Fault THEN
		sSm.sm_timeout:=TRUE;
		fb_state_entry.i16_next_step := FEHLER;

	ELSIF
		sCtrl.in.Warning AND NotausOK THEN
		sSm.sm_Error_Warnung:=TRUE;
		fb_state_entry.i16_next_step := FEHLER;

	ELSIF
		fb_state_entry.i16_next_step >= BEREIT AND
		sCtrl.in.Fault THEN
		sSm.sm_Error_Klemme:=TRUE;
		fb_state_entry.i16_next_step := FEHLER;

	ELSIF
		fb_state_entry.i16_next_step >= BEREIT AND
		NOT Connect THEN
		sSm.sm_connect:=TRUE;
		fb_state_entry.i16_next_step := FEHLER;

	ELSIF
		sConfig.ModeOfOperation = CSV AND
		sFb.ton_uez_velo.Q THEN
		sSm.sm_Check_Velo:=TRUE;
	(*	stop:=TRUE;*)

(*	ELSIF fb_state_entry.i16_next_step >= BEREIT AND  sConfig.UeberlaufControl_on AND
		sPos.i32_count_ueberlauf <> 0 THEN
		sSm.sm_Ueberlauf:=TRUE;
		fb_state_entry.i16_next_step := FEHLER;*)
	ELSIF fb_state_entry.i16_next_step >= BEREIT AND  sConfig.Torque_Limit >0 AND
		sConfig.Torque_Limit > e_Torque THEN
		sSm.sm_Torque_zu_gross:=TRUE;
		fb_state_entry.i16_next_step := FEHLER;

	ELSIF sConfig.ModeOfOperation = CSP AND
		sPos.lr_MaxDiff > sConfig.max_PosDiff AND
		sConfig.PosDiffControl_on THEN
		sSm.sm_PosDiff:=TRUE;
		stop:=TRUE;
	END_IF
END_IF

(* ==================================Schrittkette================================ *)
fb_state_entry(	i16_pos:= 1);

CASE fb_state_entry.i16_step OF
(*=======================================================*)
INIT_OBJ:
	fb_state_entry.i16_next_step := INIT;

(*==========================================================================================================*)
INIT:
	IF	 fb_state_entry.E THEN

		sFb.ton_uez.IN := FALSE;
		sFb.ton_quitt.IN := FALSE;
		Stop:=FALSE;
		Reset:=FALSE;
		Busy:=FALSE;
		Error_:=FALSE;
		Done:=FALSE;
		Ready:=FALSE;
		on:=FALSE;

		sCtrl.out:=sCtrlEmpty.out;

	END_IF

		IF	sConfig.aktiv THEN
			fb_state_entry.i16_next_step := 20;
		ELSE
			fb_state_entry.i16_next_step := INAKTIV;
		END_IF

20:(*Switched_on*)

	IF	fb_state_entry.E THEN
		sCtrl.out.Fault_reset:=TRUE;
		sFb.ton_uez.IN:=TRUE;
	END_IF

	(*-----------------------Weiterschaltbedingungen----------------------------*)

	IF	NOT sCtrl.in.Fault THEN
		fb_state_entry.i16_next_step := BEREIT;
		sCtrl.out.Fault_reset:=FALSE;
	ELSE
		IF	sFb.ton_uez.Q THEN
			fb_state_entry.i16_next_step := FEHLER;
		END_IF
	END_IF

(*==========================================================================================================*)
BEREIT:
	IF	fb_state_entry.E THEN
		sFb.ton_uez.IN:=FALSE;
		Ready:=TRUE;
	END_IF

	IF	(sFb.r_trig_MotorOn.Q OR MotorOn)AND
		NOT on THEN
		IF 	NotausOK THEN
			MotorOn:=FALSE;
			sCtrl.out.Target_Position:=sCtrl.in.Position;
			fb_state_entry.i16_next_step := 110;
		ELSE
			sSm.sm_NotausNok:=TRUE;
			fb_state_entry.i16_next_step := FEHLER;
		END_IF
	END_IF

	CASE	sConfig.ModeOfOperation OF

	CSV:
			;
	CSP:
		(*Positionsübergabe*)

		IF 	on AND
			(*Positive Richtung*)
			 ((sVisuAxis.BtnJogP.Pressed AND sVisuAxis.b_kont) OR MoveP) THEN
			IF	sConfig.SW_Limit_on THEN
				IF	sCtrl.in.Position < sConfig.SW_Limit_max THEN
					sCtrl.out.Target_Position:=sConfig.SW_Limit_max;
				END_IF
			ELSE
				sCtrl.out.Target_Position:=sCtrl.in.Position+10000;
			END_IF
			Busy:=TRUE;
			Done:=FALSE;
		END_IF

		IF 	on AND
			(*Negative Richtung*)
			((sVisuAxis.BtnJogM.Pressed AND sVisuAxis.b_kont) OR MoveN) THEN
			IF	sConfig.SW_Limit_on THEN
				IF	sCtrl.in.Position > sConfig.SW_Limit_min THEN
					sCtrl.out.Target_Position:=sConfig.SW_Limit_min;
				END_IF
			ELSE
				sCtrl.out.Target_Position:=sCtrl.in.Position-10000;
			END_IF
			Busy:=TRUE;
			Done:=FALSE;
		END_IF

		(*Jog beenden*)
		IF	sFb.r_trig_jogP.Q OR sFb.r_trig_jogM.Q OR
			sFb.r_trig_MoveP.Q OR sFb.r_trig_MoveM.Q OR
			sFb.r_trig_stop.Q OR reset OR
			Stop  THEN
			Busy:=FALSE;
			Done:=TRUE;
			MoveP:=FALSE;
			MoveN:=FALSE;
			sCtrl.out.Target_Position:=sCtrl.in.Position;
		END_IF


		(*Positionieren mit Positionsvorgabe Absolut*)
		IF	on  AND
			(sFb.r_trig_MoveAbs.Q OR MoveAbs)THEN
			IF	sConfig.SW_Limit_on THEN
				IF	Vorgabe_Pos_Abs > sConfig.SW_Limit_max THEN
					sCtrl.out.Target_Position:=sConfig.SW_Limit_max;
					sSm.sm_SW_Limit:=TRUE;
				ELSIF	Vorgabe_Pos_Abs < sConfig.SW_Limit_min THEN
					sCtrl.out.Target_Position:=sConfig.SW_Limit_min;
					sSm.sm_SW_Limit:=TRUE;
				ELSE
					sCtrl.out.Target_Position:=Vorgabe_Pos_Abs;
					sSm.sm_SW_Limit:=FALSE;
				END_IF
			ELSE
				sCtrl.out.Target_Position:=Vorgabe_Pos_Abs;
			END_IF
			Busy:=TRUE;
			Done:=FALSE;
			bMove:=TRUE;
		END_IF

		(*Positionieren mit Positionsvorgabe Relativ*)
		IF	on  AND
			MoveRel THEN
			IF	sConfig.SW_Limit_on THEN
				IF	Vorgabe_Pos_Rel+sCtrl.out.Target_Position > sConfig.SW_Limit_max THEN
					sCtrl.out.Target_Position:=sConfig.SW_Limit_max;
					sSm.sm_SW_Limit:=TRUE;
				ELSIF	Vorgabe_Pos_Rel+sCtrl.out.Target_Position < sConfig.SW_Limit_min THEN
					sCtrl.out.Target_Position:=sConfig.SW_Limit_min;
					sSm.sm_SW_Limit:=TRUE;
				ELSE
					sCtrl.out.Target_Position:=sCtrl.out.Target_Position+Vorgabe_Pos_Rel;
					sSm.sm_SW_Limit:=FALSE;
				END_IF
			ELSE
				sCtrl.out.Target_Position:=sCtrl.out.Target_Position+Vorgabe_Pos_Rel;
			END_IF
			Busy:=TRUE;
			Done:=FALSE;
			bMove:=TRUE;
		END_IF
		IF	NOT on  AND
			(MoveAbs OR MoveRel)THEN
			fb_state_entry.i16_next_step := FEHLER;
		END_IF
	END_CASE

	(*Regler abschalten*)
	IF	(sFb.r_trig_reset.Q OR MotorOff OR NOT NotausOK )AND
		on	THEN
		sSm.sm_Move:=bMove;
		fb_state_entry.i16_next_step := 210;
	END_IF

	sFb.ton_Busy(IN:=Busy , PT:= t#50ms, Q=> , ET=> );
	IF	sFb.ton_Busy.Q AND On_Position AND
		fb_state_entry.i16_next_step = fb_state_entry.i16_step THEN
		Busy:=FALSE;
		Done:=TRUE;
		bMove:=FALSE;
		IF	sSm.sm_SW_Limit THEN
			fb_state_entry.i16_next_step := FEHLER;
		END_IF
	END_IF

	MotorOff:=FALSE;
	Stop:=FALSE;
	MoveAbs:=FALSE;
	MoveRel:=FALSE;

	IF	fb_state_entry.X THEN
		sFb.ton_uez.IN:=TRUE;
		Busy:=TRUE;
		Error_:=FALSE;
		Done:=FALSE;
		bMove:=FALSE;
	END_IF

(*==========================================================================================================*)
110:(*Ready_to_switch_on*)

	IF	fb_state_entry.E THEN
		sCtrl.out.Enable_voltage:=TRUE;
		sCtrl.out.Shutdown:=TRUE;
		sSm:=sSmEmpty;
	END_IF

	(*-----------------------Weiterschaltbedingungen----------------------------*)
	IF	sCtrl.in.Ready_to_switch_on THEN
		sCtrl.out.Switch_on:=TRUE;
		fb_state_entry.i16_next_step := 120;
	END_IF

(*=======================================================*)
120:(*Switched_on*)

	IF	fb_state_entry.E THEN
		sCtrl.out.Switch_on:=TRUE;
	END_IF

	(*-----------------------Weiterschaltbedingungen----------------------------*)

	IF	sCtrl.in.Switched_on THEN
		fb_state_entry.i16_next_step := 130;
	END_IF

130:(*Operation_enabled*)

	IF	fb_state_entry.E THEN
		sCtrl.out.Enable_operation:=TRUE;
	END_IF

	(*-----------------------Weiterschaltbedingungen----------------------------*)

	IF	sCtrl.in.Operation_enabled THEN
		fb_state_entry.i16_next_step := BEREIT;
		Busy:=FALSE;
		Error_:=FALSE;
		on:=TRUE;
	END_IF

(*==========================================================================================================*)
210:(*Switch_off*)

	IF	fb_state_entry.E THEN
		sCtrl.out.Target_Position:=sCtrl.in.Position;
		sCtrl.out.Enable_operation:=FALSE;
		sCtrl.out.Switch_on:=FALSE;
		on:=FALSE;
		MoveP:=FALSE;
		MoveN:=FALSE;
		Reset:=FALSE;
	END_IF

	(*-----------------------Weiterschaltbedingungen----------------------------*)

	IF	NOT sCtrl.in.Operation_enabled THEN
			fb_state_entry.i16_next_step := 220;
	END_IF

(*=======================================================*)
220:(*Shutdown*)

	IF	fb_state_entry.E THEN
		sCtrl.out.Shutdown:=FALSE;
	END_IF

	(*-----------------------Weiterschaltbedingungen----------------------------*)

	IF	NOT sCtrl.in.Ready_to_switch_on THEN
		fb_state_entry.i16_next_step := 230;
	END_IF

230:(*disabled_voltage*)

	IF	fb_state_entry.E THEN
			sCtrl.out.Enable_voltage:=FALSE;
	END_IF

	(*-----------------------Weiterschaltbedingungen----------------------------*)

	IF	sCtrl.in.Switch_on_disabled THEN
		sCtrl.out.Target_Position:=sCtrl.in.Position;
		fb_state_entry.i16_next_step := 240;
		Busy:=FALSE;
		Error_:=FALSE;
	END_IF

240:(**)
	IF	sSm.sm_PosDiff OR
		sSm.sm_Check_Velo OR
		sSm.sm_Move THEN
		fb_state_entry.i16_next_step := FEHLER;
	ELSE
		fb_state_entry.i16_next_step := BEREIT;
		sSm:=sSmEmpty;
	END_IF

(*==========================================================================================================*)
FEHLER: (*Fehler*)
	IF	fb_state_entry.E THEN
		Busy:=FALSE;
		Error_:=TRUE;
		Ready:=FALSE;
		on:=FALSE;
		MoveP:=FALSE;
		MoveN:=FALSE;
		sCtrl.out:=sCtrlEmpty.out;

		IF	sSm.sm_timeout THEN
			FB_ReadXmlLineMsg.ID:='sm_timeout';
			Error.No:=1;
		ELSIF	sSm.sm_Error_Klemme THEN
			FB_ReadXmlLineMsg.ID:='sm_Error_Klemme';
			Error.No:=2;
		ELSIF	sSm.sm_Error_Warnung THEN
			FB_ReadXmlLineMsg.ID:='sm_Error_Warnung';
			Error.No:=3;
		ELSIF	sSm.sm_Check_Velo THEN
			FB_ReadXmlLineMsg.ID:='sm_Check_Velo';
			Error.No:=4;
		ELSIF	sSm.sm_SW_Limit THEN
			FB_ReadXmlLineMsg.ID:='sm_SW_Limit';
			Error.No:=5;
		ELSIF		sSm.sm_PosDiff THEN
			FB_ReadXmlLineMsg.ID:='sm_PosDiff';
			Error.No:=6;
		ELSIF		sSm.sm_fehler_daten_schreiben THEN
			FB_ReadXmlLineMsg.ID:='sm_fehler_daten_schreiben';
			Error.No:=7;
		ELSIF		sSm.sm_connect THEN
			FB_ReadXmlLineMsg.ID:='sm_connect';
			Error.No:=8;
		ELSIF		sSm.sm_Ueberlauf THEN
			FB_ReadXmlLineMsg.ID:='sm_Ueberlauf';
			Error.No:=9;
		ELSIF			sSm.sm_Torque_zu_gross THEN
			FB_ReadXmlLineMsg.ID:='sm_Torque_zu_gross';
			Error.No:=10;
		ELSIF
			sSm.sm_NotausNok	THEN
			FB_ReadXmlLineMsg.ID:='sm_NotausNok';
			Error.No:=11;
		ELSIF
			sSm.sm_Move	THEN
			FB_ReadXmlLineMsg.ID:='sm_Move';
			Error.No:=12;
		END_IF

		Error.DateTime:=gVarDTSystemtime;

	END_IF

	sVisu.ProcessTime:=ProcessTime;

	IF	sFb.r_trig_quitt.Q THEN
			fb_state_entry.i16_next_step := INIT;
	END_IF

	IF sFb.ton_quitt.Q THEN
		sFb.ton_quitt(IN := FALSE);
	END_IF

INAKTIV:

	Busy:=FALSE;
	Ready := TRUE;
	Done := TRUE;

	IF	sConfig.aktiv THEN
		fb_state_entry.i16_next_step := FEHLER;
	END_IF

END_CASE

fb_state_entry(i16_pos:= 2);


(*------------------------------------------------------------------
	Error-Handling
  ------------------------------------------------------------------*)
IF	sVisuAxis.BtnReset.Pressed OR Reset THEN
	sSm:=sSmEmpty;
END_IF
IF	(MEMCMP(ADR(sSmEmpty), ADR(sSm), SIZEOF(sSmEmpty)) = 0 ) THEN
	Error.No:=0;
	Error.Text:='';
	TempErrorText:='';
END_IF
IF Error.Text<>''	AND ST_Lng.b_EndChangeLng THEN
	(*Error.DateTime:=;*)
	Error.Typ:=0;
	ErrorHandler.AddError(ErrorToAdd:=Error,
						sVisu:=Visu.ErrorHandler);
END_IF

IF	TempErrorText <>'' AND
	FIND(TempErrorText,'#')=0 AND
	LEN(TempErrorText)>40 THEN
	TempErrorText:=CONCAT(TempErrorText, '##');
END_IF

	LaufschriftObj(
	N:= 40,
	StepWidth:=1,
	PT:= t#100ms ,
	Text:= TempErrorText,
	Display=>sVisu.ErrorString );

	LaufschriftErrh(
	N:= 100,
	StepWidth:=1,
	PT:= t#100ms ,
	Text:= TempErrorText,
	Display=>Error.Text );

FB_ReadXmlLineConf(
	Prefix:= 'CONFIG',
	ID:= sConfig.InstName,
	File:= 'CONFIG.xml',
	Text=>  );

FB_ReadXmlLineMsg(
	Prefix:= 'MSG',
	ID:= ,
	File:= 'MSG.xml',
	Text=>);

IF	Error_ THEN
	TempErrorText:=CONCAT(sConfig.InstName,': ');
(*	TempErrorText:=CONCAT(TempErrorText,sConfig.Description);*)
	TempErrorText:=CONCAT(TempErrorText,FB_ReadXmlLineConf.Text);
	TempErrorText:=CONCAT(TempErrorText,' -> ');
	TempErrorText:=CONCAT(TempErrorText,FB_ReadXmlLineMsg.Text);
END_IF
END_FUNCTION_BLOCK
ACTION Btn_init:
(*Einheiten			===============================================================================*)
IF 	sConfig.Modulo THEN
	sVisuAxis.Einheit_pos:='°';
	sVisuAxis.Einheit_velo:='rpm ';
ELSE
	sVisuAxis.Einheit_pos:='mm';
	sVisuAxis.Einheit_velo:='mm/min';
END_IF
(*===================================================================================================*)

sVisuAxis.BtnReset.Text := 'Reset / Off';
sVisuAxis.BtnReset.Enable :=  ModeSelect.Mode <=MODE_MANUAL;
sVisuAxis.BtnReset.Visible := TRUE;
IF	sVisuAxis.BtnReset.Enable THEN
	sVisuAxis.BtnReset.TextColor := Color.black;
ELSE
	sVisuAxis.BtnReset.TextColor := Color.grey;
END_IF
IF	sVisuAxis.BtnReset.Pressed THEN
	sVisuAxis.BtnReset.BackgroundColor:=Color.darkgrey;
ELSE
	sVisuAxis.BtnReset.BackgroundColor:=Color.lightgrey;
END_IF
(*-------------------------------------------------------*)
sVisuAxis.BtnStop.Text := 'Stop';
sVisuAxis.BtnStop.Enable := On AND NOT Error_ AND NOT On_Position AND ModeSelect.Mode <=MODE_MANUAL ;
sVisuAxis.BtnStop.Visible := On AND NOT Error_ AND NOT On_Position AND ModeSelect.Mode <=MODE_MANUAL AND NOT sVisuAxis.BtnJogP.Pressed AND NOT sVisuAxis.BtnJogM.Pressed;
IF	sVisuAxis.BtnStop.Enable THEN
	sVisuAxis.BtnStop.TextColor := Color.black;
ELSE
	sVisuAxis.BtnStop.TextColor := Color.grey;
END_IF
IF	sVisuAxis.BtnStop.Pressed THEN
	sVisuAxis.BtnStop.BackgroundColor:=Color.darkgrey;
ELSE
	sVisuAxis.BtnStop.BackgroundColor:=Color.lightgrey;
END_IF
(*-------------------------------------------------------*)
sVisuAxis.BtnJogP.Text := '+';
sVisuAxis.BtnJogP.Enable := On AND (On_Position OR sVisuAxis.BtnJogP.Pressed) AND NOT Error_ AND ModeSelect.Mode <=MODE_MANUAL ;
IF	sVisuAxis.BtnJogP.Enable THEN
	sVisuAxis.BtnJogP.TextColor := Color.black;
ELSE
	sVisuAxis.BtnJogP.TextColor := Color.grey;
END_IF
sVisuAxis.BtnJogP.Visible := sConfig.ModeOfOperation=CSP;
IF	sVisuAxis.BtnJogP.Pressed THEN
	sVisuAxis.BtnJogP.BackgroundColor:=Color.yellow;
ELSE
	sVisuAxis.BtnJogP.BackgroundColor:=Color.lightgrey;
END_IF
(*-------------------------------------------------------*)
sVisuAxis.BtnJogM.Text := '-';
sVisuAxis.BtnJogM.Enable := On AND (On_Position OR sVisuAxis.BtnJogM.Pressed) AND NOT Error_ AND ModeSelect.Mode <=MODE_MANUAL ;
IF	sVisuAxis.BtnJogM.Enable THEN
	sVisuAxis.BtnJogM.TextColor := Color.black;
ELSE
	sVisuAxis.BtnJogM.TextColor := Color.grey;
END_IF
sVisuAxis.BtnJogM.Visible := sConfig.ModeOfOperation=CSP;
IF	sVisuAxis.BtnJogM.Pressed THEN
	sVisuAxis.BtnJogM.BackgroundColor:=Color.yellow;
ELSE
	sVisuAxis.BtnJogM.BackgroundColor:=Color.lightgrey;
END_IF
(*-------------------------------------------------------*)
sVisuAxis.BtnMotorOn.Text := 'Motor On';
sVisuAxis.BtnMotorOn.Enable := NOT On AND NOT Error_ AND ModeSelect.Mode <=MODE_MANUAL ;
IF	sVisuAxis.BtnMotorOn.Enable THEN
	sVisuAxis.BtnMotorOn.TextColor := Color.black;
ELSE
	sVisuAxis.BtnMotorOn.TextColor := Color.grey;
END_IF
sVisuAxis.BtnMotorOn.Visible := sConfig.ModeOfOperation=CSP;
IF	sVisuAxis.BtnMotorOn.Pressed THEN
	sVisuAxis.BtnMotorOn.BackgroundColor:=Color.darkgrey;
ELSE
	sVisuAxis.BtnMotorOn.BackgroundColor:=Color.lightgrey;
END_IF

(*-------------------------------------------------------*)
sVisuAxis.BtnMoveAbs.Text := 'Move Absolut';
sVisuAxis.BtnMoveAbs.Enable :=On AND On_Position AND NOT Error_ AND Vorgabe_Pos_Abs<>sCtrl.out.Target_Position  AND ModeSelect.Mode <=MODE_MANUAL ;
IF	sVisuAxis.BtnMoveAbs.Enable THEN
	sVisuAxis.BtnMoveAbs.TextColor := Color.black;
ELSE
	sVisuAxis.BtnMoveAbs.TextColor := Color.grey;
END_IF
sVisuAxis.BtnMoveAbs.Visible := sConfig.ModeOfOperation=CSP;
IF	sVisuAxis.BtnMoveAbs.Pressed THEN
	sVisuAxis.BtnMoveAbs.BackgroundColor:=Color.yellow;
ELSE
	sVisuAxis.BtnMoveAbs.BackgroundColor:=Color.lightgrey;
END_IF

(*-------------------------------------------------------*)
sVisuAxis.BtnTeach.Text := 'Teach';
sVisuAxis.BtnTeach.Enable :=On AND NOT Error_ AND On_Position  AND ModeSelect.Mode <=MODE_MANUAL ;
IF	sVisuAxis.BtnTeach.Enable THEN
	sVisuAxis.BtnTeach.TextColor := Color.black;
ELSE
	sVisuAxis.BtnTeach.TextColor := Color.grey;
END_IF
sVisuAxis.BtnTeach.Visible := sConfig.ModeOfOperation=CSP;
IF	sVisuAxis.BtnTeach.Pressed THEN
	sVisuAxis.BtnTeach.BackgroundColor:=Color.grey;
ELSE
	sVisuAxis.BtnTeach.BackgroundColor:=Color.lightgrey;
END_IF
END_ACTION
ACTION Description:
;(*======================================================
   FB: fb_72x1_Achse (Achse ohne NC verfahren)
 ------------------------------------------------------
   Auth: 		Werner Friedl    						 
   Date: 		18.04.2018   						     
   Rev.: 		1.0	
   Desc:		Mit diesem FB  können Antriebe ohne NC mit der PLC verfahren werden.
			- Die Struktur "sConfig" beinhaltet alle Variablen zur Motorkonfiguration.
			- über die VAR_INPUT	kann die Achse positioniert werden.
			  und über VAR_OUTPUT kann der Zustand abgefragt werden.
			  Beschreibung (siehe Variablendeklaration)	

			- Motor Bereit zum Einschalten: Ready
	
			- Motor einschalten:		MotorOn:=TRUE;
			- Motor ausschalten:  	MotorOff:=TRUE;

			- Abragen ob eingeschaltet:	On

--->			- Relative Bewegung (inkremental)
				Bewegung starten:	MoveRel:=TRUE; 
									Vorgabe_Pos_Rel:=100;
									Vorgabe_Velo:=1000;
				Bewegung gestartet:	Busy    
				Position erreicht :	Done

-->			- Absolute Bewegung
				Bewegung starten:	MoveAbs:=TRUE; 
									Vorgabe_Pos_Abs:=100;
									Vorgabe_Velo:=1000;
				Bewegung gestartet:	Busy    
				Position erreicht :	Done

-->			- Motor bewegen ohne Positionierung
			  (Softwarelimit abschalten sonst fährt die Achse nur bis zum Limit): 
									MoveP:=TRUE;	(positiv)
									MoveN:=TRUE	(negativ)
									Vorgabe_Velo:=1000;

				Bewegung gestartet:	Busy

	- Die Zählrichtunug des Messsystem wird im tsm eingestellt (Coe-Online 8000.01 
	- Die Globale CONSTANTE 	NO_OF_POS_AXIS  beschreibt die Anzahl der Positinen in der Positionsliste.
    	- in den TD kann eine Positionsliste angelegt werden. z.B.	
		TD.Posxxxxx	 			: ARRAY [1..NO_OF_POS_AXIS] OF st_Pos;	
	- in den MP muss ein PosOffset und ein Override angelegt werden.
		MP.xxxx.PosOffset_xxxx	 		: st_Pos;
		MP.xxxx.Override_xxxx			: DINT :=10;
	- für diesen FB gibt es ein Visuobjekt: 	ZLIB_7211_ACHSE
	- alle Strukturen im Ordner EL72x1 müssen vorhanden sein



